METHOD PUBLIC DoPlanning : BOOL
VAR_INPUT
	count : UDINT;
END_VAR
VAR
	i, j  : INT;
END_VAR
IF count = 0 THEN
	isFinished := FALSE;
	Initialize();
END_IF

IF RequireRepeateBlegCenter=TRUE AND BlegCenterFinished=TRUE AND state=BlegCenter THEN
	state:=ready;
    RequireBlegCenter:=TRUE;
	RequireRepeateBlegCenter:=FALSE;
END_IF
IF RequireRepeateStoneRot=TRUE AND StoneRotFinished=TRUE AND state=StoneRot THEN
	state:=MlegRollB;
    MlegRollBFinished:=TRUE;
    RequireStoneRot:=TRUE;
	RequireRepeateStoneRot:=FALSE;
END_IF

IF RequireRepeateBodyPosAdjust=TRUE AND state=BodyPosAdjust AND BodyPosAdjustFinished=TRUE THEN
	state:=ReduceHeight;
    ReduceHeightFinished:=TRUE; 
	RequireBodyPosAdjust:=TRUE;
	RequireRepeateBodyPosAdjust:=FALSE;
END_IF
IF RequireRepeateBLegPosAdjust=TRUE AND state=BLegPosAdjust AND BLegPosAdjustFinished=TRUE THEN
	state:=BodyPosAdjust;
    BodyPosAdjustFinished:=TRUE; 
	RequireBLegPosAdjust:=TRUE;
	RequireRepeateBLegPosAdjust:=FALSE;
END_IF

IF RequireRepeateSearchPedal=TRUE AND state=SearchPedal AND SearchPedalFinished=TRUE THEN
	state:=BLegPosAdjust;
    BLegPosAdjustFinished:=TRUE; 
	RequireSearchPedal:=TRUE;
	RequireRepeateSearchPedal:=FALSE;
END_IF

IF RequireRepeateArmControl=TRUE AND state=ArmControl AND ArmControlFinished=TRUE THEN
	state:=SearchPedal;
    SearchPedalFinished:=TRUE; 
	RequireArmControl:=TRUE;
	RequireRepeateArmControl:=FALSE;
END_IF

IF RequireRepeateOrientAdjust=TRUE AND state=OrientAdjust AND OrientAdjustFinished=TRUE THEN
	state:=ArmControl;
    ArmControlFinished:=TRUE; 
	RequireOrientAdjust:=TRUE;
	RequireRepeateOrientAdjust:=FALSE;
END_IF

StateMachine();
TrjPlanning();

IF quit_flag THEN
	isFinished := TRUE;
	quit_flag := FALSE;
	AC_visual_start:=AC_visual_start;
	
RequireAddHeightFromWalk:=FALSE;
RequireBlegCenter:=FALSE;
RequireMlegRollA:=FALSE;
RequireFlegRotA:=FALSE;
RequireReduceHeight:=FALSE;	
RequireBodyPosAdjust:=FALSE;
RequireBLegPosAdjust:=FALSE;
RequireSearchPedal:=FALSE;
RequireArmControl:=FALSE;
RequireOrientAdjust:=FALSE;
RequireMlegRollB:=FALSE;	
RequireStoneRot:=FALSE;		
RequireLiftMleg:=FALSE;
RequireSpeedUp:=FALSE;
RequireSlide:=FALSE;
RequirePushReleaseBall:=FALSE;
RequireSpeedDown:=FALSE;
RequireBLegRecovery:=FALSE;
RequireMlegRollC:=FALSE;
RequireAddHeight:=FALSE;
RequireFlegRotB:=FALSE;
RequireRecovery:=FALSE;
RequireReduceHeightB:=FALSE;

AddHeightFromWalkFinished:=FALSE;
BlegCenterFinished:=FALSE;
MlegRollAFinished:=FALSE;
FlegRotAFinished:=FALSE;
ReduceHeightFinished:=FALSE;
BodyPosAdjustFinished:=FALSE;
BLegPosAdjustFinished:=FALSE;
SearchPedalFinished:=FALSE;
ArmControlFinished:=FALSE;
OrientAdjustFinished:=FALSE;
MlegRollBFinished:=FALSE;
StoneRotFinished:=FALSE;
LiftMlegFinished:=FALSE;
SpeedUpFinished:=FALSE;
SlideFinished:=FALSE;
PushReleaseBallFinished:=FALSE;
SpeedDownFinished:=FALSE;
BLegRecoveryFinished:=FALSE;
MlegRollCFinished:=FALSE;
AddHeightFinished:=FALSE;
FlegRotBFinished:=FALSE;
CurlingGaitFinished:=FALSE;
RecoveryFinished:=FALSE;
ReduceHeightBFinished:=FALSE;
ReadyFinished:=FALSE;
IsCurlingFinished:=FALSE;
CurlingGaitFinished:=FALSE;
	
	RequireRepeateBlegCenter:=FALSE;
	RequireRepeateBodyPosAdjust:=FALSE;
	RequireRepeateSearchPedal:=FALSE;
	RequireRepeateBLegPosAdjust:=FALSE;
	RequireRepeateOrientAdjust:=FALSE;
	RequireRepeateStoneRot:=FALSE;
END_IF
END_METHOD

METHOD PUBLIC Initialize : BOOL
VAR_INPUT
END_VAR
VAR
	i, j : INT;
	
	leg_pos    : ARRAY[0..2] OF LREAL;
	
	Rb : Mat3;
	hip_pos_j  : Vec3;
	leg_pos_wrt_com : Vec3;
	
END_VAR
Rleg[0]:=SetMat3(1,0,0,0,0,-1,0,1,0);
Rleg[1]:=SetMat3(-1,0,0,0,0,1,0,1,0,);
Rleg[2]:=SetMat3(-1,0,0,0,0,1,0,1,0);
Rleg[3]:=SetMat3(-1,0,0,0,0,1,0,1,0);
Rleg[4]:=SetMat3( -1,0,0,0,0,1,0,1,0);
Rleg[5]:=SetMat3(1,0,0,0,0,-1,0,1,0);

state:=Ready;
ReadyFinished:=true;
quit_flag  := FALSE;
gait_cycle := 0;
AC_visual_start:=FALSE;

IF gvl.taskChooseId=0 THEN //击打
	gvl.target_vel_init:=2;
	gvl.PushVelocityIn_init:=2.3;
	gvl.stone_rot_vel_init:=-60;
	gvl.slideTimeIn_init:=0.3;
	gvl.PushFinishDurationTimeIn_init:=1;
ELSE //进营
	gvl.target_vel_init:=2;
	gvl.PushVelocityIn_init:=1.15;
	gvl.stone_rot_vel_init:=30;	
	gvl.slideTimeIn_init:=0.3;
	gvl.PushFinishDurationTimeIn_init:=1;
END_IF

gvl.adjust_angle_degree:=gvl.adjust_angle_degree_init;
gvl.target_vel:=gvl.target_vel_init;
gvl.stone_rot_vel:=gvl.stone_rot_vel_init;//rpm
gvl.PushVelocityIn:=gvl.PushVelocityIn_init;
gvl.BPA_adjust_angle_degree:=gvl.BPA_adjust_angle_degree_init;//degree
gvl.BPA_adjust_x:=gvl.BPA_adjust_x_init;
gvl.BPA_adjust_y:=gvl.BPA_adjust_y_init;
gvl.BLPA_adjust_distance_desire:=gvl.BLPA_adjust_distance_desire_init;	
gvl.curlingPushModel:=gvl.curlingPushModel_init;	
gvl.PushFinishDurationTimeIn:=gvl.PushFinishDurationTimeIn_init;
gvl.slideTimeIn:=gvl.slideTimeIn_init;
gvl.ArmRetractControl:=gvl.ArmRetractControl_init;
gvl.AC_AngleDegIn:=gvl.AC_AngleDegIn_init;	

// control button for each state, need be commented out at actual environment
RequireAddHeightFromWalk:=FALSE;
RequireBlegCenter:=FALSE;
RequireMlegRollA:=FALSE;
RequireFlegRotA:=FALSE;
RequireReduceHeight:=FALSE;	
RequireBodyPosAdjust:=FALSE;
RequireBLegPosAdjust:=FALSE;
RequireSearchPedal:=FALSE;
RequireArmControl:=FALSE;
RequireOrientAdjust:=FALSE;
RequireMlegRollB:=FALSE;	
RequireStoneRot:=FALSE;		
RequireLiftMleg:=FALSE;
RequireSpeedUp:=FALSE;
RequireSlide:=FALSE;
RequirePushReleaseBall:=FALSE;
RequireSpeedDown:=FALSE;
RequireBLegRecovery:=FALSE;
RequireMlegRollC:=FALSE;
RequireAddHeight:=FALSE;
RequireFlegRotB:=FALSE;
RequireRecovery:=FALSE;
RequireReduceHeightB:=FALSE;

AddHeightFromWalkFinished:=FALSE;
BlegCenterFinished:=FALSE;
MlegRollAFinished:=FALSE;
FlegRotAFinished:=FALSE;
ReduceHeightFinished:=FALSE;
BodyPosAdjustFinished:=FALSE;
BLegPosAdjustFinished:=FALSE;
SearchPedalFinished:=FALSE;
ArmControlFinished:=FALSE;
OrientAdjustFinished:=FALSE;
MlegRollBFinished:=FALSE;
StoneRotFinished:=FALSE;
LiftMlegFinished:=FALSE;
SpeedUpFinished:=FALSE;
SlideFinished:=FALSE;
PushReleaseBallFinished:=FALSE;
SpeedDownFinished:=FALSE;
BLegRecoveryFinished:=FALSE;
MlegRollCFinished:=FALSE;
AddHeightFinished:=FALSE;
FlegRotBFinished:=FALSE;
CurlingGaitFinished:=FALSE;
RecoveryFinished:=FALSE;
ReduceHeightBFinished:=FALSE;

RequireRepeateBlegCenter:=FALSE;
RequireRepeateBodyPosAdjust:=FALSE;
RequireRepeateBLegPosAdjust:=FALSE;
RequireRepeateSearchPedal:=FALSE;
RequireRepeateArmControl:=FALSE;
RequireRepeateOrientAdjust:=FALSE;
RequireRepeateStoneRot:=FALSE;

// bodyRot
delta_t:=1.0/gvl.SampleRate;//sample time
SetTargetValue(GVL.adjust_angle_degree,GVL.target_vel,GVL.stone_rot_vel);
IsReady:=true;

FOR i := 0 TO 5 DO
	FOR j := 0 TO 2 DO
		(*IF ABS(gvl.jntLastRefPos[i, j] - gvl.jntActualPos[i, j]) < gvl.curling_threshold_value THEN
			joint_ref_pos_init[i].data[j] := gvl.jntLastRefPos[i, j];
		ELSE
			joint_ref_pos_init[i].data[j] := gvl.jntActualPos[i, j];
		END_IF*)
		joint_ref_pos_init[i].data[j] := gvl.jntLastRefPos[i, j];
		jointPosLast[i,j]:=joint_ref_pos_init[i].data[j];
	END_FOR
END_FOR

sum_height := 0;
FOR j := 0 TO 5 DO
	// FK
	gvl.legCtrl[j].ForwardKinetics(motorAngles := joint_ref_pos_init[j].data, legIndex:=j, tipPosition => leg_pos);
	leg_ref_pos_init_wrt_hip[j] := SetVec3(leg_pos[0], leg_pos[1], leg_pos[2]);
	sum_height := sum_height - leg_ref_pos_init_wrt_hip[j].data[1];
END_FOR
body_ref_pos_init := SetVec3(0, 0, sum_height/6.0);
body_ref_ang_init := SetVec3(0, 0, 0);                            

FOR j := 0 TO 5 DO
	fbRotMat(yaw := body_ref_ang_init.data[2],
             pitch := body_ref_ang_init.data[1],
             roll := body_ref_ang_init.data[0],
             rm => Rb );
	hip_pos_j := SetVec3(hip_pos[j, 0], hip_pos[j, 1], hip_pos[j, 2]);
	leg_pos_wrt_com := VecAdd(MatMulVec(Rleg[j], leg_ref_pos_init_wrt_hip[j]), hip_pos_j);
    leg_ref_pos_init[j] := VecAdd(body_ref_pos_init, MatMulVec(Rb, leg_pos_wrt_com));
END_FOR

body_ref_pos := body_ref_pos_init;
body_ref_ang := body_ref_ang_init;
leg_ref_pos := leg_ref_pos_init;
leg_ref_pos_wrt_hip := leg_ref_pos_init_wrt_hip;
leg_ref_pos_last:=leg_ref_pos;

FOR i := 0 TO 5 DO
	FOR j := 0 TO 2 DO
		jointPosTarget[i, j] := joint_ref_pos_init[i].data[j];
		jointVelTarget[i, j] := 0;
		jointFceTarget[i, j] := 0;
	END_FOR
END_FOR
END_METHOD

METHOD PUBLIC isPedal : BOOL
VAR_INPUT
		legIndex:INT;
END_VAR
IF ABS(gvl.tipActualFce[legIndex,0])>30 THEN //10 need be calibrated40-->35
	isPedal:=TRUE;
ELSE
	isPedal:=FALSE;
END_IF
END_METHOD

METHOD PUBLIC isStone : BOOL
VAR_INPUT
	legIndex:INT;
END_VAR
IF ABS(gvl.tipActualFce[legIndex,2])>50 THEN //10 need be calibrated
	isStone:=TRUE;
ELSE
	isStone:=FALSE;
END_IF
END_METHOD

METHOD PUBLIC SetTargetValue : BOOL
VAR_INPUT
	in_adjust_angle_degree:LREAL:=0;//unit:degree
	in_target_vel:LREAL:=0;//unit:m/s
	in_stone_rot_vel:LREAL:=0;//unit:rpm
END_VAR
adjust_angle_rad:=in_adjust_angle_degree*pi/180;
target_vel:=in_target_vel;
stone_rot_vel:=in_stone_rot_vel/60*2*pi;
END_METHOD

METHOD PUBLIC StateMachine : BOOL
VAR_INPUT
END_VAR

VAR
	i: INT;
	j: INT;
	RotRadius: LREAL;
END_VAR
IF state=ready AND RequireAddHeightFromWalk=TRUE THEN
	state:=AddHeightFromWalk;
	IsReady:=FALSE;
	IsAddHeightFromWalk:=TRUE;
	RequireAddHeightFromWalk:=FALSE;
	body_ref_pos_enter := body_ref_pos;
	body_ref_ang_enter := body_ref_ang;
	leg_ref_pos_enter := leg_ref_pos;
	EnterAddHeightFromWalkCount:=gait_cycle;
	AddHeightFromWalkFinished:=FALSE;
	AHFW_body_target_pos:=body_ref_pos_enter;
	AHFW_body_target_pos.data[2]:=AHFW_body_target_pos.data[2]+compensateDistance;	

ELSIF state=AddHeightFromWalk AND RequireBlegCenter=TRUE THEN
	state:=BlegCenter;
	IsAddHeightFromWalk:=FALSE;
	IsBlegCenter:=TRUE;
	RequireBlegCenter:=FALSE;
	body_ref_pos_enter := body_ref_pos;
	body_ref_ang_enter := body_ref_ang;
	leg_ref_pos_enter := leg_ref_pos;
	EnterBlegCenterCount:=gait_cycle;
	IsLeg0Move:=TRUE;
	BlegCenterFinished:=FALSE;
	FOR i:=0 TO 1 DO
		FOR j:=0 TO 2 DO
			BlegCenter_BJntStart[i].data[j]:=jointPosLast[Mapping05[i],j];
		END_FOR
	END_FOR
ELSIF state=BlegCenter AND BlegCenterFinished=TRUE AND RequireMlegRollA=TRUE THEN
	state:=MlegRollA;
	IsBlegCenter:=FALSE;
	IsMlegRollA:=TRUE;
	requireMlegRollA:=FALSE;
	body_ref_pos_enter := body_ref_pos;
	body_ref_ang_enter := body_ref_ang;
	leg_ref_pos_enter := leg_ref_pos;
	EnterMlegRollACount:=gait_cycle;
	MlegRollAFinished:=FALSE;
	FOR i:=0 TO 1 DO
		FOR j:=0 TO 2 DO
			MlegRollA_MJntStart[i].data[j]:=jointPosLast[Mapping14[i],j];
		END_FOR
	END_FOR
ELSIF state=MlegRollA AND MlegRollAFinished=TRUE AND RequireFlegRotA=TRUE THEN
	state:=FlegRotA;
	IsMlegRollA:=FALSE;
	IsFlegRotA:=TRUE;
	requireFlegRotA:=FALSE;
	body_ref_pos_enter := body_ref_pos;
	body_ref_ang_enter := body_ref_ang;
	leg_ref_pos_enter := leg_ref_pos;
	EnterFlegRotACount:=gait_cycle;
	FlegRotAFinished:=FALSE;
	FOR i:=0 TO 1 DO
		FOR j:=0 TO 2 DO
			FlegRotA_FJntStart[i].data[j]:=jointPosLast[Mapping23[i],j];
		END_FOR
	END_FOR
ELSIF state=FlegRotA AND FlegRotAFinished=TRUE AND RequireReduceHeight=TRUE THEN
	state:=ReduceHeight;
	IsFlegRotA:=FALSE;
	IsReduceHeight:=TRUE;
	requireReduceHeight:=FALSE;
	body_ref_pos_enter := body_ref_pos;
	body_ref_ang_enter := body_ref_ang;
	leg_ref_pos_enter := leg_ref_pos;
	EnterReduceHeightCount:=gait_cycle;
	body_target_pos:=body_ref_pos_enter;
	body_target_pos.data[2]:=targetHeight;
	ReduceHeightFinished:=FALSE;
	FOR i:=0 TO 1 DO
		FOR j:=0 TO 2 DO
			ReduceHeight_FJntRef[i].data[j]:=jointPosLast[Mapping23[i],j];
		END_FOR
	END_FOR
ELSIF state=ReduceHeight AND ReduceHeightFinished=TRUE AND RequireBodyPosAdjust=TRUE THEN
	state:=BodyPosAdjust;
	IsReduceHeight:=FALSE;
	IsBodyPosAdjust:=TRUE;
	requireBodyPosAdjust:=FALSE;
	body_ref_pos_enter := body_ref_pos;
	body_ref_ang_enter := body_ref_ang;
	leg_ref_pos_enter := leg_ref_pos;
	EnterBodyPosAdjustCount:=gait_cycle;
	BodyPosAdjustFinished:=FALSE;		
	FOR i:=0 TO 1 DO
		FOR j:=0 TO 2 DO
			BPA_FJntRef[i].data[j]:=jointPosLast[Mapping23[i],j];
			BPA_MJntExtend[i,j]:=jointPosLast[Mapping14[i],j];
			BPA_BJntExtend[i,j]:=jointPosLast[Mapping05[i],j];
		END_FOR
		BPA_MJntExtract[i,0]:=BPA_MJntExtend[i,0];
		BPA_MJntExtract[i,1]:=BPA_MJntExtend[i,1]-10*pi/180.0;
		BPA_MJntExtract[i,2]:=BPA_MJntExtend[i,2]+10*pi/180.0;
		BPA_BJntExtract[i,0]:=BPA_BJntExtend[i,0];
		BPA_BJntExtract[i,1]:=BPA_BJntExtend[i,1]-10*pi/180.0;
		BPA_BJntExtract[i,2]:=BPA_BJntExtend[i,2]+10*pi/180.0;
	END_FOR	
	FOR i:=0 TO 2 DO
		BPA_RotCenter1.data[i]:=0.5*(leg_ref_pos_enter[0].data[i]+leg_ref_pos_enter[5].data[i]);
	END_FOR	
	BPA_BodyPosStart:=body_ref_pos_enter;
	BPA_BodyAngStart:=body_ref_ang_enter;	
	RotRadius:=SQRT((BPA_BodyPosStart.data[0]-BPA_RotCenter1.data[0])*(BPA_BodyPosStart.data[0]-BPA_RotCenter1.data[0])+
				(BPA_BodyPosStart.data[1]-BPA_RotCenter1.data[1])*(BPA_BodyPosStart.data[1]-BPA_RotCenter1.data[1]));	
	BPA_AngRad:=GVL.BPA_adjust_angle_degree*pi/180;
	BPA_x:=gvl.BPA_adjust_x;
	BPA_y:=gvl.BPA_adjust_y;
	BPA_BodyPoseEnd.data[0]:=BPA_RotCenter1.data[0]+RotRadius*COS(BPA_AngRad+BPA_BodyAngStart.data[2])+BPA_x;
	BPA_BodyPoseEnd.data[1]:=BPA_RotCenter1.data[1]+RotRadius*SIN(BPA_AngRad+BPA_BodyAngStart.data[2])+BPA_y;
	BPA_BodyPoseEnd.data[2]:=body_ref_pos_enter.data[2];
	BPA_BodyAngEnd:=BPA_BodyAngStart;
	BPA_BodyAngEnd.data[2]:=BPA_BodyAngStart.data[2]+BPA_AngRad;	
ELSIF state=BodyPosAdjust AND BodyPosAdjustFinished=TRUE AND RequireBLegPosAdjust=TRUE THEN
	state:=BLegPosAdjust;
	IsBodyPosAdjust:=FALSE;
	IsBLegPosAdjust:=TRUE;
	requireBLegPosAdjust:=FALSE;
	body_ref_pos_enter := body_ref_pos;
	body_ref_ang_enter := body_ref_ang;
	leg_ref_pos_enter := leg_ref_pos;
	EnterBLegPosAdjustCount:=gait_cycle;
	BLegPosAdjustFinished:=FALSE;	
	
	BLPA_tgtLegPos:=leg_ref_pos_enter;
	BLPA_adjust_distance:=gvl.BLPA_adjust_distance_desire;
	FOR i:=0 TO 1 DO
		FOR j:=0 TO 1 DO
			BLPA_tgtLegPos[Mapping05[i]].data[j]:=leg_ref_pos_enter[Mapping05[i]].data[j]+BLPA_adjust_distance[i,j];
		END_FOR
	END_FOR
	
ELSIF state=BLegPosAdjust AND BLegPosAdjustFinished=TRUE AND RequireSearchPedal=TRUE THEN
	state:=SearchPedal;
	IsBLegPosAdjust:=FALSE;
	IsSearchPedal:=TRUE;
	requireSearchPedal:=FALSE;
	body_ref_pos_enter := body_ref_pos;
	body_ref_ang_enter := body_ref_ang;
	leg_ref_pos_enter := leg_ref_pos;
	EnterSearchPedalCount:=gait_cycle;
	SearchPedalFinished:=FALSE;	
	SP_RBLegSearching:=TRUE;SP_LBLegSearching:=FALSE;
	SP_BLegSearchFinished[0]:=FALSE;SP_BLegSearchFinished[1]:=FALSE;
	SP_PedalSearched[0]:=FALSE;SP_PedalSearched[1]:=FALSE;
	SP_EnterSubSearchCount[0]:=gait_cycle;SP_EnterSubSearchCount[1]:=gait_cycle;
	SP_EnterSubSearchDecreaseCount[0]:=gait_cycle;SP_EnterSubSearchDecreaseCount[1]:=gait_cycle;
	FOR i:=0 TO 1 DO
		FOR j:=0 TO 2 DO
			SP_BJntStart[i].data[j]:=jointPosLast[Mapping05[i],j];
		END_FOR
		gvl.legCtrl[Mapping05[i]].ForwardKinetics(motorAngles:=SP_BJntStart[i].data , legIndex:=Mapping05[i] , tipPosition=>SP_BPosStartWrtHip[i].data );
	END_FOR
ELSIF state=SearchPedal AND SearchPedalFinished=TRUE AND RequireArmControl=TRUE THEN
	state:=ArmControl;
	IsSearchPedal:=FALSE;
	IsArmControl:=TRUE;
	requireArmControl:=FALSE;
	body_ref_pos_enter := body_ref_pos;
	body_ref_ang_enter := body_ref_ang;
	leg_ref_pos_enter := leg_ref_pos;
	EnterArmControlCount:=gait_cycle;
	ArmControlFinished:=FALSE;	
	
	AC_AngleDeg:=gvl.AC_AngleDegIn;
	AC_AngleRad:=AC_AngleDeg*pi/180;
	AC_Velocity:=AC_AngleRad/AC_time;
	AC_extend:=TRUE;
	AC_retract:=FALSE;
	AC_wait:=FALSE;
	AC_EnterExtendCount:=gait_cycle;
	AC_EnterRetractCount:=gait_cycle;
	AC_visual_start:=false;
	

ELSIF state=ArmControl AND ArmControlFinished=TRUE AND RequireOrientAdjust=TRUE THEN
	state:=OrientAdjust;
	IsArmControl:=FALSE;
	IsOrientAdjust:=TRUE;
	requireOrientAdjust:=FALSE;
	body_ref_pos_enter := body_ref_pos;
	body_ref_ang_enter := body_ref_ang;
	leg_ref_pos_enter := leg_ref_pos;
	EnterOrientAdjustCount:=gait_cycle;
	OrientAdjustFinished:=FALSE;	
	FOR i:=0 TO 1 DO
		FOR j:=0 TO 2 DO
			OA_FJntRef[i].data[j]:=jointPosLast[Mapping23[i],j];
			OA_MJntExtend[i,j]:=jointPosLast[Mapping14[i],j];
		END_FOR
		OA_MJntExtract[i,0]:=OA_MJntExtend[i,0];
		OA_MJntExtract[i,1]:=OA_MJntExtend[i,1]-10*pi/180.0;
		OA_MJntExtract[i,2]:=OA_MJntExtend[i,2]+10*pi/180.0;
	END_FOR
	FOR i:=0 TO 2 DO
		OA_RotCenter1.data[i]:=0.5*(leg_ref_pos_enter[0].data[i]+leg_ref_pos_enter[5].data[i]);
	END_FOR
	OA_BodyPosStart:=body_ref_pos_enter;
	OA_BodyAngStart:=body_ref_ang_enter;
	RotRadius:=SQRT((OA_BodyPosStart.data[0]-OA_RotCenter1.data[0])*(OA_BodyPosStart.data[0]-OA_RotCenter1.data[0])+
               (OA_BodyPosStart.data[1]-OA_RotCenter1.data[1])*(OA_BodyPosStart.data[1]-OA_RotCenter1.data[1]));
	adjust_angle_rad:=GVL.adjust_angle_degree*pi/180;
	OA_BodyPoseEnd.data[0]:=OA_RotCenter1.data[0]+RotRadius*COS(adjust_angle_rad+OA_BodyAngStart.data[2]);
	OA_BodyPoseEnd.data[1]:=OA_RotCenter1.data[1]+RotRadius*SIN(adjust_angle_rad+OA_BodyAngStart.data[2]);
	OA_BodyPoseEnd.data[2]:=body_ref_pos_enter.data[2];
	OA_BodyAngEnd:=OA_BodyAngStart;
	OA_BodyAngEnd.data[2]:=OA_BodyAngStart.data[2]+adjust_angle_rad;
ELSIF state=OrientAdjust AND OrientAdjustFinished=TRUE AND RequireMlegRollB=TRUE THEN
	state:=MlegRollB;
	IsOrientAdjust:=FALSE;
	IsMlegRollB:=TRUE;
	requireMlegRollB:=FALSE;
	body_ref_pos_enter := body_ref_pos;
	body_ref_ang_enter := body_ref_ang;
	leg_ref_pos_enter := leg_ref_pos;
	EnterMlegRollBCount:=gait_cycle;
	FOR i:=0 TO 1 DO
		FOR j:=0 TO 2 DO
			MlegRollB_MJntStart[i].data[j]:=jointPosLast[Mapping14[i],j];
		END_FOR
	END_FOR	
ELSIF state=MlegRollB AND MlegRollBFinished=TRUE AND RequireStoneRot=TRUE THEN
	state:=StoneRot;
	stone_rot_vel:=GVL.stone_rot_vel/60*2*pi;
	IsMlegRollB:=FALSE;
	IsStoneRot:=TRUE;
	requireStoneRot:=FALSE;
	body_ref_pos_enter := body_ref_pos;
	body_ref_ang_enter := body_ref_ang;
	leg_ref_pos_enter := leg_ref_pos;
	EnterStoneRotCount:=gait_cycle;
	StoneRotFinished:=FALSE;
	SetColide:=FALSE;
	StoneRotSubState[0]:=FALSE;
	StoneRotSubState[1]:=FALSE;
	FOR i:=0 TO 1 DO
		FOR j:=0 TO 2 DO
			StoneRot_FJntStart[i].data[j]:=jointPosLast[Mapping23[i],j];
		END_FOR
	END_FOR
ELSIF state=StoneRot AND StoneRotFinished=TRUE AND  RequireLiftMleg=TRUE THEN
	state:=LiftMleg;
	IsStoneRot:=FALSE;
	IsLiftMleg:=TRUE;
	requireLiftMleg:=FALSE;	
	body_ref_pos_enter := body_ref_pos;
	body_ref_ang_enter := body_ref_ang;
	leg_ref_pos_enter := leg_ref_pos;
	EnterLiftMlegCount:=gait_cycle;
	LiftMlegFinished:=FALSE;
	FOR i:=0 TO 1 DO
		FOR j:=0 TO 2 DO
			LiftMleg_MJntStart[i].data[j]:=jointPosLast[Mapping14[i],j];
		END_FOR
	END_FOR	
ELSIF state=LiftMleg AND LiftMlegFinished=TRUE AND RequireSpeedUp=TRUE THEN
	state:=SpeedUp;
	IsLiftMleg:=FALSE;
	IsSpeedUp:=TRUE;
	requireSpeedUp:=FALSE;	
	IF ABS(GVL.target_vel)<=0.5 THEN
		GVL.target_vel:=0.5;
	END_IF
	target_vel:=GVL.target_vel;
	body_ref_pos_enter := body_ref_pos;
	body_ref_ang_enter := body_ref_ang;
	leg_ref_pos_enter := leg_ref_pos;
	EnterSpeedUpCount:=gait_cycle;
	SpeedUpFinished:=FALSE;
	FOR i:=0 TO 1 DO
		FOR j:=0 TO 2 DO
			SpeedUp_MJntRef[i].data[j]:=jointPosLast[Mapping14[i],j];
			SpeedUp_FJntRef[i].data[j]:=jointPosLast[Mapping23[i],j];
			SpeedUp_BJntStart[i].data[j]:=jointPosLast[Mapping05[i],j];
		END_FOR
		gvl.legCtrl[Mapping05[i]].ForwardKinetics(motorAngles:=SpeedUp_BJntStart[i].data , legIndex:=Mapping05[i] , tipPosition=>SpeedUp_BPosWrtHipStart[i].data );
	END_FOR	
	CurrentBLegMaxDistance:=MAX(ABS(SpeedUp_BPosWrtHipStart[0].data[0]),ABS(SpeedUp_BPosWrtHipStart[1].data[0]));
	Distance_x_total:=0.85-CurrentBLegMaxDistance;
	IF Distance_x_total<0 THEN
		quit_flag:=TRUE;
		SpeedUpFinished:=true;
	END_IF
	
	SpeedUpSubState:=SpeedUpAS;
	EnterSpeedUpASCount:=gait_cycle;

	Distance_x_AS:=Distance_x_total-Distance_x_DS-target_vel*Time_CS;
	Time_AS:=2.0*Distance_x_AS/target_vel;
ELSIF state=SpeedUp AND SpeedUpFinished=TRUE AND RequireSlide=TRUE THEN
	state:=Slide;
	IsSpeedUp:=FALSE;
	IsSlide:=TRUE;
	requireSlide:=FALSE;	
	body_ref_pos_enter := body_ref_pos;
	body_ref_ang_enter := body_ref_ang;
	leg_ref_pos_enter := leg_ref_pos;
	EnterSlideCount:=gait_cycle;
	SlideFinished:=FALSE;
	slideTime:=gvl.slideTimeIn;
ELSIF state=Slide AND SlideFinished=TRUE AND RequirePushReleaseBall=TRUE THEN
	state:=PushReleaseBall;
	IsSlide:=FALSE;
	IsPushReleaseBall:=TRUE;
	RequirePushReleaseBall:=FALSE;
	body_ref_pos_enter := body_ref_pos;
	body_ref_ang_enter := body_ref_ang;
	leg_ref_pos_enter := leg_ref_pos;
	EnterPushReleaseBallCount:=gait_cycle;
	PushReleaseBallFinished:=FALSE;
	PushFinishDurationTime:=gvl.PushFinishDurationTimeIn;
	FOR i:=0 TO 1 DO
		FOR j:=0 TO 2 DO
			PushReleaseBall_FJntStart[i].data[j]:=jointPosLast[Mapping23[i],j];
		END_FOR
		gvl.legCtrl[Mapping23[i]].ForwardKinetics(motorAngles:=PushReleaseBall_FJntStart[i].data , legIndex:=Mapping23[i] , tipPosition=>PushReleaseBall_FPosStartWrtHip[i].data );
	END_FOR
	IF ABS(gvl.PushVelocityIn)<=0.1 THEN
		gvl.PushVelocityIn:=0;
	END_IF
	PushVelocity:=gvl.PushVelocityIn;
	PushDistance:=PRDistance_x_total-DecVelDistance-PRConstVelTime*PushVelocity;
	PRConstVelDistance:=PRConstVelTime*PushVelocity;
	PushTime:=PushDistance*2/PushVelocity;
	
ELSIF state=PushReleaseBall AND PushReleaseBallFinished=TRUE AND RequireSpeedDown=TRUE THEN
	state:=SpeedDown;
	IsPushReleaseBall:=FALSE;
	IsSpeedDown:=TRUE;
	RequireSpeedDown:=FALSE;
	body_ref_pos_enter := body_ref_pos;
	body_ref_ang_enter := body_ref_ang;
	leg_ref_pos_enter := leg_ref_pos;
	EnterSpeedDownCount:=gait_cycle;
	SpeedDownFinished:=FALSE;
	FOR i:=0 TO 1 DO
		FOR j:=0 TO 2 DO
			SpeedDown_MJntStart[i].data[j]:=jointPosLast[Mapping14[i],j];
		END_FOR
	END_FOR
ELSIF state=SpeedDown AND SpeedDownFinished=TRUE AND RequireBLegRecovery=TRUE THEN	
	state:=BLegRecovery;
	IsSpeedDown:=FALSE;
	IsBLegRecovery:=TRUE;
	RequireBLegRecovery:=FALSE;
	body_ref_pos_enter := body_ref_pos;
	body_ref_ang_enter := body_ref_ang;
	leg_ref_pos_enter := leg_ref_pos;
	EnterBLegRecoveryCount:=gait_cycle;
	BLegRecoveryFinished:=FALSE;	
	FOR i:=0 TO 1 DO
		FOR j:=0 TO 2 DO
			BLR_FJntStart[i].data[j]:=jointPosLast[Mapping05[i],j];
		END_FOR
	END_FOR
	
ELSIF state=BLegRecovery AND BLegRecoveryFinished=TRUE AND RequireMlegRollC=TRUE THEN
	state:=MlegRollC;
	IsBLegRecovery:=FALSE;
	IsMlegRollC:=TRUE;
	RequireMlegRollC:=FALSE;
	body_ref_pos_enter := body_ref_pos;
	body_ref_ang_enter := body_ref_ang;
	leg_ref_pos_enter := leg_ref_pos;
	EnterMlegRollCCount:=gait_cycle;
	MlegRollCFinished:=FALSE;	
	FOR i:=0 TO 1 DO
		FOR j:=0 TO 2 DO
			MlegRollC_MJntStart[i].data[j]:=jointPosLast[Mapping14[i],j];
		END_FOR
	END_FOR
ELSIF state=MlegRollC AND MlegRollCFinished=TRUE AND RequireAddHeight=TRUE THEN	
	state:=AddHeight;
	RequireAddHeight:=FALSE;
	IsMlegRollC:=FALSE;
	IsAddHeight:=TRUE;
	body_ref_pos_enter := body_ref_pos;
	body_ref_ang_enter := body_ref_ang;
	leg_ref_pos_enter := leg_ref_pos;
	EnterAddHeightCount:=gait_cycle;
	AddHeightFinished:=FALSE;
	FOR i:=0 TO 1 DO
		FOR j:=0 TO 2 DO
			AddHeight_FJntStart[i].data[j]:=jointPosLast[Mapping23[i],j];
		END_FOR
	END_FOR
	body_target_pos:=body_ref_pos_enter;
	body_target_pos.data[2]:=sum_height/6.0+compensateDistance;
ELSIF state=AddHeight AND AddHeightFinished=TRUE AND RequireFlegRotB=TRUE THEN	
	state:=FlegRotB;
	IsAddHeight:=FALSE;
	IsFlegRotB:=TRUE;
	RequireFlegRotB:=FALSE;
	body_ref_pos_enter := body_ref_pos;
	body_ref_ang_enter := body_ref_ang;
	leg_ref_pos_enter := leg_ref_pos;
	EnterFlegRotBCount:=gait_cycle;
	FlegRotBFinished:=FALSE;
	FOR i:=0 TO 1 DO
		FOR j:=0 TO 2 DO
			FlegRotB_FJntStart[i].data[j]:=jointPosLast[Mapping23[i],j];
		END_FOR
	END_FOR
ELSIF state=FlegRotB AND FlegRotBFinished=TRUE AND RequireRecovery=TRUE THEN	
	state:=Recovery;
	IsFlegRotB:=FALSE;
	IsRecovery:=TRUE;
	RequireRecovery:=FALSE;	
	body_ref_pos_enter := body_ref_pos;
	body_ref_ang_enter := body_ref_ang;
	leg_ref_pos_enter := leg_ref_pos;
	EnterRecoveryCount:=gait_cycle;
	RecoveryFinished:=FALSE;	
	RcJointPosStart:=jointPosLast;
	
ELSIF state=Recovery AND RecoveryFinished=TRUE AND RequireReduceHeightB=TRUE THEN	
	state:=ReduceHeightB;
	IsRecovery:=FALSE;
	IsReduceHeightB:=TRUE;
	RequireReduceHeightB:=FALSE;	
	body_ref_pos_enter := body_ref_pos;
	body_ref_ang_enter := body_ref_ang;
	leg_ref_pos_enter := leg_ref_pos;
	EnterReduceHeightBCount:=gait_cycle;
	ReduceHeightBFinished:=FALSE;	
	RHB_body_target_pos:=body_ref_pos_enter;
	RHB_body_target_pos.data[2]:=RHB_body_target_pos.data[2]-compensateDistance;

ELSIF state=ReduceHeightB AND ReduceHeightBFinished=TRUE THEN	
	IsReduceHeightB:=FALSE;
	IsCurlingFinished:=TRUE;
	state:=CurlingFinished;
	CurlingGaitFinished:=TRUE;
	quit_flag:=TRUE;
END_IF
END_METHOD

METHOD PUBLIC TrjPlanning : BOOL
VAR_INPUT
END_VAR
VAR
	tr : LREAL;
	i, j : INT;
	Rb : Mat3;
	hip_pos_j : Vec3;
	leg_ref_pos_wrt_com_j : Vec3;
	tmp : Vec3;
	tip_pos, tip_vel : Vec3;
	
	body_ref_pos_start : Vec3;
	body_ref_pos_end : Vec3;
	jointTmpPosLast: ARRAY[0..2] OF LREAL;
	body_ref_ang_start: Vec3;
	leg_ref_pos_start: ARRAY [0..5] OF Vec3;
	leg_ref_pos_target: ARRAY [0..5] OF Vec3;
	body_ref_ang_end: Vec3;
	Rb_target2: Mat3;
	Rb_target1: Mat3;
	leg_ref_pos_end: ARRAY [0..5] OF Vec3;
	fbElipseInterpolation:ElipseInterpolation;
	fbHermitInterpolation:HermitInterpolation;
	
	tempTipForce:ARRAY [0..2] OF LREAL;
	temJntActPos:ARRAY [0..2] OF LREAL;
	tempDesJntTrq:ARRAY [0..2] OF LREAL;
END_VAR
gait_cycle := gait_cycle + 1;

IF state=Ready THEN
	body_ref_pos := body_ref_pos_init;
	body_ref_ang := body_ref_ang_init;
	leg_ref_pos := leg_ref_pos_init;
	leg_ref_pos_wrt_hip := leg_ref_pos_init_wrt_hip;
ELSIF state=AddHeightFromWalk THEN
	TrjPlanning_AddHeightFromWalk();
ELSIF state=BlegCenter THEN
	TrjPlanning_BlegCenter();
ELSIF state=MlegRollA THEN
	TrjPlanning_MlegRollA();
ELSIF state=FlegRotA THEN
	TrjPlanning_FlegRotA();
ELSIF state=ReduceHeight THEN
	TrjPlanning_ReduceHeight();
ELSIF state=BodyPosAdjust THEN
	TrjPlanning_BodyPosAdjust();
ELSIF state=BLegPosAdjust THEN
	TrjPlanning_BLegPosAdjust();	
ELSIF state=SearchPedal THEN
	TrjPlanning_SearchPedal();
ELSIF state=ArmControl THEN
	TrjPlanning_ArmControl();
ELSIF state=OrientAdjust THEN	
	TrjPlanning_OrientAdjust();
ELSIF state=MlegRollB THEN
	TrjPlanning_MlegRollB();
ELSIF state=StoneRot THEN
	TrjPlanning_StoneRot();
ELSIF state=LiftMleg THEN
	TrjPlanning_LiftMleg();
ELSIF state=SpeedUp THEN
	TrjPlanning_SpeedUp();
ELSIF state=Slide THEN	
	TrjPlanning_Slide();
ELSIF state=PushReleaseBall THEN
	TrjPlanning_PushReleaseBall();
ELSIF state=SpeedDown THEN	
	TrjPlanning_SpeedDown();
ELSIF state=BLegRecovery THEN	
	TrjPlanning_BLegRecovery();
ELSIF state=MlegRollC THEN	
	TrjPlanning_MlegRollC();
ELSIF state=AddHeight THEN	
	TrjPlanning_AddHeight();
ELSIF state=FlegRotB THEN	
	TrjPlanning_FlegRotB();
ELSIF state=Recovery THEN	
	TrjPlanning_Recovery();	
ELSIF state=ReduceHeightB THEN	
	TrjPlanning_ReduceHeightB();	
END_IF

// transform TO leg local frame AND DO inverse kinematics

FOR j := 0 TO 5 DO
	fbRotMat(
    	yaw := body_ref_ang.data[2], 
		pitch := body_ref_ang.data[1], 
		roll := body_ref_ang.data[0], 
		rm => Rb);
	hip_pos_j := SetVec3(hip_pos[j, 0], hip_pos[j, 1], hip_pos[j, 2]);

	//leg_ref_pos_wrt_com = Rb' * (leg_ref_pos - body_ref_pos)
	leg_ref_pos_wrt_com_j := MatMulVec(
		                         MatTranspose(Rb),
								 VecAdd(
									 leg_ref_pos[j],
									 VecNeg(body_ref_pos)
                                 )
                             );
	// leg_ref_pos_wrt_hip = Rleg' * (leg_ref_pos_wrt_com_j - hip_pos)
	leg_ref_pos_next_wrt_hip[j] := MatMulVec(
		                               MatTranspose(Rleg[j]),
									   VecAdd(
										   leg_ref_pos_wrt_com_j,
										   VecNeg(hip_pos_j)
									   )
								   );
								   
	leg_ref_vel_next_wrt_hip[j] := VecMulNum(VecAdd(leg_ref_pos_next_wrt_hip[j], VecNeg(leg_ref_pos_wrt_hip[j])), DINT_TO_LREAL(gvl.sampleRate));
END_FOR


// mapping to actual joints
FOR j := 0 TO 5 DO
	tmp := leg_ref_pos_next_wrt_hip[leg_index_mapping[j]-1];
	tip_pos := SetVec3(tmp.data[0], tmp.data[1], tmp.data[2]);
	tmp := leg_ref_vel_next_wrt_hip[leg_index_mapping[j]-1];
	tip_vel := SetVec3(tmp.data[0], tmp.data[1], tmp.data[2]);
	FOR i:= 0 TO 2 DO
		jointTmpPosLast[i]:=jointPosLast[j,i];
	END_FOR		
	gvl.legCtrl[j].InversePosAndVel(
		tipPos := tip_pos.data, 
		tipVel := tip_vel.data, 
		refPosLast:=jointTmpPosLast,
		legIndex:=j,
		jntPos => joint_ref_pos[j].data, 
		jntVel => joint_ref_vel[j].data);
	
END_FOR

//generate joint reference torque
FOR i:=0 TO 5 DO
	tempTipForce[0]:=tipForceDesire[i,0];tempTipForce[1]:=tipForceDesire[i,1];tempTipForce[2]:=tipForceDesire[i,2];
	temJntActPos[0]:=gvl.jntActualPos[i,0];temJntActPos[1]:=gvl.jntActualPos[i,1];temJntActPos[2]:=gvl.jntActualPos[i,2];
	gvl.legCtrl[i].DesireDriveForce(fTipDes:=tempTipForce , motorAng:=temJntActPos , legIndex:=i , fDrvDes=>tempDesJntTrq );
	jntTrqDesire[i,0]:=tempDesJntTrq[0];jntTrqDesire[i,1]:=tempDesJntTrq[1];jntTrqDesire[i,2]:=tempDesJntTrq[2];
END_FOR


// link to physical outputs
FOR i := 0 TO 5 DO
	FOR j := 0 TO 2 DO
		jointPosTarget[i, j] := joint_ref_pos[i].data[j];
		jointPosLast[i,j]:=jointPosTarget[i, j] ;
		gvl.jntRefPosLastPlanning[i,j]:=jointPosTarget[i, j] ;
		jointVelTarget[i, j] := joint_ref_vel[i].data[j];
		jointFceTarget[i, j] :=jntTrqDesire[i,j];
	END_FOR
END_FOR

// store refs for next loop
leg_ref_pos_wrt_hip := leg_ref_pos_next_wrt_hip;
leg_ref_pos_last:=leg_ref_pos;

IF gait_cycle > tTotalAll * gvl.sampleRate THEN
	quit_flag := TRUE;
END_IF
END_METHOD

METHOD PUBLIC TrjPlanning_AddHeight : BOOL
VAR_INPUT
END_VAR
VAR
	tr: LREAL;
	i: INT;
	Rb_target1: Mat3;
	temp:vec3;
END_VAR
IF  AddHeightFinished=FALSE AND (gait_cycle-EnterAddHeightCount)<=AddHeightTime*gvl.sampleRate THEN
	body_ref_ang:=body_ref_ang_enter;
	leg_ref_pos:=leg_ref_pos_enter;
	tr  := UDINT_TO_LREAL(gait_cycle - EnterAddHeightCount) / gvl.sampleRate / AddHeightTime;
	fbGetPivot(tNow := tr, tTotal := 1.0, pivot => pvt);
	FOR i:=0 TO 2 DO
		body_ref_pos.data[i]:=(1-pvt)*body_ref_pos_enter.data[i]+pvt*body_target_pos.data[i];
	END_FOR
	
	FOR i:=0 TO 1 DO
		gvl.legCtrl[Mapping23[i]].ForwardKinetics(motorAngles:=AddHeight_FJntStart[i].data , legIndex:=Mapping23[i] , tipPosition=>AddHeight_FPosWrtHip[i].data );
		fbRotMat(yaw := body_ref_ang_enter.data[2], pitch := body_ref_ang_enter.data[1],roll := body_ref_ang_enter.data[0], rm => Rb_target1 );
		temp.data[0]:=hip_pos[Mapping23[i],0];temp.data[1]:=hip_pos[Mapping23[i],1];temp.data[2]:=hip_pos[Mapping23[i],2];
		leg_ref_pos[Mapping23[i]]:= VecAdd( MatMulVec(Rb_target1, VecAdd(temp,MatMulVec(Rleg[Mapping23[i]],AddHeight_FPosWrtHip[i]))),body_ref_pos);
	END_FOR
ELSE
	AddHeightFinished:=TRUE;	
	RequireFlegRotB:=TRUE;//********************************************************************************************************
END_IF
END_METHOD

METHOD PUBLIC TrjPlanning_AddHeightFromWalk : BOOL
VAR_INPUT
END_VAR
VAR
	tr: LREAL;
	i: INT;
	Rb_target1: Mat3;
	temp: vec3;
END_VAR
IF AddHeightFromWalkFinished=FALSE AND (gait_cycle-EnterAddHeightFromWalkCount)<=AHFW_time*gvl.sampleRate THEN
	body_ref_ang:=body_ref_ang_enter;
	leg_ref_pos:=leg_ref_pos_enter;
	tr  := UDINT_TO_LREAL(gait_cycle - EnterAddHeightFromWalkCount) / gvl.sampleRate / AHFW_time;
	fbGetPivot(tNow := tr, tTotal := 1.0, pivot => pvt);
	FOR i:=0 TO 2 DO
		body_ref_pos.data[i]:=(1-pvt)*body_ref_pos_enter.data[i]+pvt*AHFW_body_target_pos.data[i];
	END_FOR
ELSE
	AddHeightFromWalkFinished:=TRUE;
	RequireBlegCenter:=true;
END_IF
END_METHOD

METHOD PUBLIC TrjPlanning_ArmControl : BOOL
VAR_INPUT
END_VAR
IF ArmControlFinished=FALSE THEN
	body_ref_pos:=body_ref_pos_enter;
	body_ref_ang:=body_ref_ang_enter;
	leg_ref_pos:=leg_ref_pos_enter;	
	
	IF AC_extend=TRUE THEN
		AC_wait:=FALSE;
		AC_retract:=FALSE;
		IF (gait_cycle-AC_EnterExtendCount)=1 THEN
			GVL.jogVelocity[20]:=AC_Velocity;
			GVL.jogButton[20]:=TRUE;
		END_IF
		IF (gait_cycle-AC_EnterExtendCount)=LREAL_TO_UDINT(AC_time*gvl.sampleRate) THEN
			GVL.jogVelocity[20]:=0;
			GVL.jogButton[20]:=FALSE;
			GVL.jogStopButton[20]:=TRUE;
		END_IF
		IF (gait_cycle-AC_EnterExtendCount)=LREAL_TO_UDINT((AC_time+0.5)*gvl.sampleRate) THEN
			AC_visual_start:=TRUE;
		END_IF
		IF (gait_cycle-AC_EnterExtendCount)=LREAL_TO_UDINT((AC_time+0.5+2)*gvl.sampleRate) THEN
			AC_visual_start:=FALSE;
			gvl.ArmRetractControl:=TRUE;
		END_IF		
		
	END_IF
	
	IF AC_retract=FALSE AND gvl.ArmRetractControl=TRUE AND (gait_cycle-AC_EnterExtendCount)>=LREAL_TO_UDINT(AC_time*gvl.sampleRate) THEN
		AC_retract:=TRUE;
		AC_visual_start:=FALSE;
		gvl.ArmRetractControl:=FALSE;
		AC_EnterRetractCount:=gait_cycle;
	END_IF
	
	IF AC_retract=TRUE THEN
		AC_extend:=FALSE;
		AC_wait:=FALSE;
		IF (gait_cycle-AC_EnterRetractCount)=1 THEN
			GVL.jogVelocity[20]:=-AC_Velocity;
			GVL.jogButton[20]:=TRUE;
		END_IF	
		IF (gait_cycle-AC_EnterRetractCount)=LREAL_TO_UDINT(AC_time*gvl.sampleRate) THEN
			GVL.jogVelocity[20]:=0;
			GVL.jogButton[20]:=FALSE;
			GVL.jogStopButton[20]:=TRUE;
			ArmControlFinished:=TRUE;
		END_IF
	END_IF
END_IF
END_METHOD

METHOD PUBLIC TrjPlanning_BlegCenter : BOOL
VAR_INPUT
END_VAR
VAR

											 
	(*BC_BPosExtendRefDouble:ARRAY[0..1,0..2] OF LREAL:=[-0.15,-0.3805-0.07-0.01,0,
												       -0.15,-0.3805-0.07-0.01,0];
	BC_BPosExtendRefSingle:ARRAY[0..1,0..2] OF LREAL:=[-0.15,-0.3805-0.07-0.01,-0.05,
												       -0.15,-0.3805-0.07-0.01,0.05];											
	BC_BPosRetractRef:ARRAY[0..1,0..2]      OF LREAL:=[-0.15,-0.3805,0,
												       -0.15,-0.3805,0];*)
													   											 
	BC_BPosExtendRefDouble:ARRAY[0..1,0..2] OF LREAL:=[-0.15,-0.4-0.07-0.01,0.02*1.125,
												       -0.15,-0.4-0.07-0.01,-0.02*1.125];
	BC_BPosExtendRefSingle:ARRAY[0..1,0..2] OF LREAL:=[-0.15,-0.4-0.07-0.01,-0.05,
												       -0.15,-0.4-0.07-0.01,0.05];											
	BC_BPosRetractRef:ARRAY[0..1,0..2]      OF LREAL:=[-0.15,-0.4,0,
												       -0.15,-0.4,0];
												 
	BC_BJntRetractRef:ARRAY[0..1,0..2]      OF LREAL:=[0,180*pi/180,330*pi/180,
                                                       0,180*pi/180,330*pi/180];	
	BC_BJntTargetRef:ARRAY[0..1,0..2]       OF LREAL:=[0*pi/180,190.9254*pi/180, 312.9903*pi/180,
                                                       0*pi/180,190.9254*pi/180, 312.9903*pi/180];//double pedal,[-0.15, -0.3805-0.07-0.01,0]														 
		
	tTotal:lreal;										 
	tNow: LREAL;
	i: INT;
	j: INT;
	tr: LREAL;
	Rb_target1: Mat3;
	temp: vec3;
	tempLeg:ARRAY [0..2] OF LREAL;
	tempJnt:ARRAY [0..2] OF LREAL;
	tempRef:ARRAY [0..2] OF LREAL;
	
	tipForceDesireLegA:	 ARRAY[0..5,0..2] OF LREAL:=[0,-100,0,
													 0,0,0,
													 0,0,0,
													 0,0,0,
													 0,0,0,
													 0,0,0];
	tipForceDesireLegF:	 ARRAY[0..5,0..2] OF LREAL:=[0,0,0,
													 0,0,0,
													 0,0,0,
													 0,0,0,
													 0,0,0,
													 0,-120,0];													 
END_VAR
IF (gait_cycle-EnterBlegCenterCount)=1 THEN
	IF BlegCenterType=0 THEN
		FOR i:=0 TO 1 DO
			tempLeg[0]:=BC_BPosExtendRefDouble[i,0];tempLeg[1]:=BC_BPosExtendRefDouble[i,1];tempLeg[2]:=BC_BPosExtendRefDouble[i,2];
			tempRef[0]:=BC_BJntTargetRef[i,0];tempRef[1]:=BC_BJntTargetRef[i,1];tempRef[2]:=BC_BJntTargetRef[i,2];
			GVL.legCtrl[Mapping05[i]].InverseKinetics(tipPosition:=tempLeg , refPosLast:=tempRef , legIndex:=Mapping05[i] , motorAngles=>tempJnt , isSingular=> );
			BC_BJntTarget[i,0]:=tempJnt[0];BC_BJntTarget[i,1]:=tempJnt[1];BC_BJntTarget[i,2]:=tempJnt[2];
		END_FOR
	ELSE
		FOR i:=0 TO 1 DO
			tempLeg[0]:=BC_BPosExtendRefSingle[i,0];tempLeg[1]:=BC_BPosExtendRefSingle[i,1];tempLeg[2]:=BC_BPosExtendRefSingle[i,2];
			tempRef[0]:=BC_BJntTargetRef[i,0];tempRef[1]:=BC_BJntTargetRef[i,1];tempRef[2]:=BC_BJntTargetRef[i,2];
			GVL.legCtrl[Mapping05[i]].InverseKinetics(tipPosition:=tempLeg , refPosLast:=tempRef , legIndex:=Mapping05[i] , motorAngles=>tempJnt , isSingular=> );
			BC_BJntTarget[i,0]:=tempJnt[0];BC_BJntTarget[i,1]:=tempJnt[1];BC_BJntTarget[i,2]:=tempJnt[2];
		END_FOR
	END_IF
	FOR i:=0 TO 1 DO
		tempLeg[0]:=BC_BPosRetractRef[i,0];tempLeg[1]:=BC_BPosRetractRef[i,1];tempLeg[2]:=BC_BPosRetractRef[i,2];
		tempRef[0]:=BC_BJntRetractRef[i,0];tempRef[1]:=BC_BJntRetractRef[i,1];tempRef[2]:=BC_BJntRetractRef[i,2];
		GVL.legCtrl[Mapping05[i]].InverseKinetics(tipPosition:=tempLeg , refPosLast:=tempRef , legIndex:=Mapping05[i] , motorAngles=>tempJnt , isSingular=> );
		BC_BJntRetract[i,0]:=tempJnt[0];BC_BJntRetract[i,1]:=tempJnt[1];BC_BJntRetract[i,2]:=tempJnt[2];
	END_FOR	
END_IF

IF (gait_cycle-EnterBlegCenterCount)=(BlegCenterRetractTime+BlegCenterExtendTime)*gvl.sampleRate THEN
	leg_ref_pos_enter:=leg_ref_pos_last;
END_IF
IF IsLeg0Move=FALSE AND (gait_cycle-EnterLeg5MoveCount)=(BlegCenterRetractTime+BlegCenterExtendTime)*gvl.sampleRate THEN
	leg_ref_pos_enter:=leg_ref_pos_last;
END_IF


body_ref_pos:=body_ref_pos_enter;
body_ref_ang:=body_ref_ang_enter;
leg_ref_pos:=leg_ref_pos_enter;
IF BlegCenterFinished=FALSE THEN
	IF IsLeg0Move=TRUE THEN
		IF (gait_cycle-EnterBlegCenterCount)<=BlegCenterRetractTime*gvl.sampleRate THEN
			tr  := UDINT_TO_LREAL(gait_cycle-EnterBlegCenterCount) / gvl.sampleRate / BlegCenterRetractTime;
			fbGetPivot(tNow := tr, tTotal := 1.0, pivot => pvt);
			FOR j:=0 TO 2 DO
				BlegCenter_BJntRef[0].data[j]:=(1-pvt)*BlegCenter_BJntStart[0].data[j]+pvt*(BC_BJntRetract[0,j]);
			END_FOR		
			gvl.legCtrl[Mapping05[0]].ForwardKinetics(motorAngles:=BlegCenter_BJntRef[0].data , legIndex:=Mapping05[0] , tipPosition=>BlegCenter_BPosWrtHip[0].data );
			fbRotMat(yaw := body_ref_ang_enter.data[2], pitch := body_ref_ang_enter.data[1],roll := body_ref_ang_enter.data[0], rm =>  Rb_target1 );
			temp.data[0]:=hip_pos[Mapping05[0],0];temp.data[1]:=hip_pos[Mapping05[0],1];temp.data[2]:=hip_pos[Mapping05[0],2];
			leg_ref_pos[Mapping05[0]]:= VecAdd( MatMulVec(Rb_target1, VecAdd(temp,MatMulVec(Rleg[Mapping05[0]],BlegCenter_BPosWrtHip[0]))),body_ref_pos);
		ELSIF (gait_cycle-EnterBlegCenterCount)<=(BlegCenterRetractTime+BlegCenterExtendTime)*gvl.sampleRate THEN
			tr  := (UDINT_TO_LREAL(gait_cycle-EnterBlegCenterCount) / gvl.sampleRate -BlegCenterRetractTime)/ BlegCenterExtendTime;
			fbGetPivot(tNow := tr, tTotal := 1.0, pivot => pvt);
			FOR j:=0 TO 2 DO
				BlegCenter_BJntRef[0].data[j]:=(1-pvt)*BC_BJntRetract[0,j]+pvt*(BC_BJntTarget[0,j]);
			END_FOR
			gvl.legCtrl[Mapping05[0]].ForwardKinetics(motorAngles:=BlegCenter_BJntRef[0].data , legIndex:=Mapping05[0] , tipPosition=>BlegCenter_BPosWrtHip[0].data );
			fbRotMat(yaw := body_ref_ang_enter.data[2], pitch := body_ref_ang_enter.data[1],roll := body_ref_ang_enter.data[0], rm =>  Rb_target1 );
			temp.data[0]:=hip_pos[Mapping05[0],0];temp.data[1]:=hip_pos[Mapping05[0],1];temp.data[2]:=hip_pos[Mapping05[0],2];
			leg_ref_pos[Mapping05[0]]:= VecAdd( MatMulVec(Rb_target1, VecAdd(temp,MatMulVec(Rleg[Mapping05[0]],BlegCenter_BPosWrtHip[0]))),body_ref_pos);	
		ELSE				
			IsLeg0Move:=FALSE;
			IsLeg5Move:=TRUE;
			EnterLeg5MoveCount:=gait_cycle;
			leg_ref_pos_enter:=leg_ref_pos_last;
		END_IF
		
		//force compensator
		tipForceTarget:=tipForceDesireLegF;
		IF (gait_cycle-EnterBlegCenterCount)<=fceLoadTime*gvl.sampleRate THEN
			tr  := UDINT_TO_LREAL(gait_cycle-EnterBlegCenterCount) / gvl.sampleRate / fceLoadTime;
			fbGetPivot(tNow := tr, tTotal := 1.0, pivot => pvt);
			FOR i:=0 TO 5 DO
				FOR j:=0 TO 2 DO
					tipForceDesire[i,j]:=(1-pvt)*tipForceDesireZeros[i,j]+pvt*tipForceTarget[i,j];
				END_FOR
			END_FOR
		ELSIF (gait_cycle-EnterBlegCenterCount)>(BlegCenterRetractTime+BlegCenterExtendTime-fceLoadTime)*gvl.sampleRate AND (gait_cycle-EnterBlegCenterCount)<=(BlegCenterRetractTime+BlegCenterExtendTime)*gvl.sampleRate THEN
			tr  := (UDINT_TO_LREAL(gait_cycle-EnterBlegCenterCount) / gvl.sampleRate -(BlegCenterRetractTime+BlegCenterExtendTime-fceLoadTime))/ fceLoadTime;
			fbGetPivot(tNow := tr, tTotal := 1.0, pivot => pvt);
			FOR i:=0 TO 5 DO
				FOR j:=0 TO 2 DO
					tipForceDesire[i,j]:=(1-pvt)*tipForceTarget[i,j]+pvt*tipForceDesireZeros[i,j];
				END_FOR
			END_FOR	
		END_IF
		
	END_IF
	
	IF IsLeg5Move=TRUE THEN
		IF (gait_cycle-EnterLeg5MoveCount)<=BlegCenterRetractTime*gvl.sampleRate THEN
			tr  := UDINT_TO_LREAL(gait_cycle-EnterLeg5MoveCount) / gvl.sampleRate / BlegCenterRetractTime;
			fbGetPivot(tNow := tr, tTotal := 1.0, pivot => pvt);
			FOR j:=0 TO 2 DO
				BlegCenter_BJntRef[1].data[j]:=(1-pvt)*BlegCenter_BJntStart[1].data[j]+pvt*(BC_BJntRetract[1,j]);
			END_FOR	
			gvl.legCtrl[Mapping05[1]].ForwardKinetics(motorAngles:=BlegCenter_BJntRef[1].data , legIndex:=Mapping05[1] , tipPosition=>BlegCenter_BPosWrtHip[1].data );
			fbRotMat(yaw := body_ref_ang_enter.data[2], pitch := body_ref_ang_enter.data[1],roll := body_ref_ang_enter.data[0], rm =>  Rb_target1 );
			temp.data[0]:=hip_pos[Mapping05[1],0];temp.data[1]:=hip_pos[Mapping05[1],1];temp.data[2]:=hip_pos[Mapping05[1],2];
			leg_ref_pos[Mapping05[1]]:= VecAdd( MatMulVec(Rb_target1, VecAdd(temp,MatMulVec(Rleg[Mapping05[1]],BlegCenter_BPosWrtHip[1]))),body_ref_pos);
		ELSIF (gait_cycle-EnterLeg5MoveCount)<=(BlegCenterRetractTime+BlegCenterExtendTime)*gvl.sampleRate THEN
			tr  := (UDINT_TO_LREAL(gait_cycle-EnterLeg5MoveCount) / gvl.sampleRate -BlegCenterRetractTime)/ BlegCenterExtendTime;
			fbGetPivot(tNow := tr, tTotal := 1.0, pivot => pvt);
			FOR j:=0 TO 2 DO
				BlegCenter_BJntRef[1].data[j]:=(1-pvt)*BC_BJntRetract[1,j]+pvt*(BC_BJntTarget[1,j]);
			END_FOR
			gvl.legCtrl[Mapping05[1]].ForwardKinetics(motorAngles:=BlegCenter_BJntRef[1].data , legIndex:=Mapping05[1] , tipPosition=>BlegCenter_BPosWrtHip[1].data );
			fbRotMat(yaw := body_ref_ang_enter.data[2], pitch := body_ref_ang_enter.data[1],roll := body_ref_ang_enter.data[0], rm =>  Rb_target1 );
			temp.data[0]:=hip_pos[Mapping05[1],0];temp.data[1]:=hip_pos[Mapping05[1],1];temp.data[2]:=hip_pos[Mapping05[1],2];
			leg_ref_pos[Mapping05[1]]:= VecAdd( MatMulVec(Rb_target1, VecAdd(temp,MatMulVec(Rleg[Mapping05[1]],BlegCenter_BPosWrtHip[1]))),body_ref_pos);
		ELSE			
			IsLeg5Move:=FALSE;
			leg_ref_pos_enter:=leg_ref_pos_last;
			BlegCenterFinished:=TRUE;
			tipForceDesire:=tipForceDesireZeros;
			RequireMlegRollA:=TRUE;//**********************************************************************************************
		END_IF
		
		//force compensator
		tipForceTarget:=tipForceDesireLegA;
		IF (gait_cycle-EnterLeg5MoveCount)<=fceLoadTime*gvl.sampleRate THEN
			tr  := UDINT_TO_LREAL(gait_cycle-EnterLeg5MoveCount) / gvl.sampleRate / fceLoadTime;
			fbGetPivot(tNow := tr, tTotal := 1.0, pivot => pvt);
			FOR i:=0 TO 5 DO
				FOR j:=0 TO 2 DO
					tipForceDesire[i,j]:=(1-pvt)*tipForceDesireZeros[i,j]+pvt*tipForceTarget[i,j];
				END_FOR
			END_FOR
		ELSIF (gait_cycle-EnterLeg5MoveCount)>(BlegCenterRetractTime+BlegCenterExtendTime-fceLoadTime)*gvl.sampleRate AND (gait_cycle-EnterLeg5MoveCount)<=(BlegCenterRetractTime+BlegCenterExtendTime)*gvl.sampleRate THEN
			tr  := (UDINT_TO_LREAL(gait_cycle-EnterLeg5MoveCount) / gvl.sampleRate -(BlegCenterRetractTime+BlegCenterExtendTime-fceLoadTime))/ fceLoadTime;
			fbGetPivot(tNow := tr, tTotal := 1.0, pivot => pvt);
			FOR i:=0 TO 5 DO
				FOR j:=0 TO 2 DO
					tipForceDesire[i,j]:=(1-pvt)*tipForceTarget[i,j]+pvt*tipForceDesireZeros[i,j];
				END_FOR
			END_FOR	
		END_IF		
	END_IF
	
END_IF
END_METHOD

METHOD PUBLIC TrjPlanning_BLegPosAdjust : BOOL
VAR_INPUT
END_VAR

VAR
	i: INT;
	
	tipForceDesireLegA:	 ARRAY[0..5,0..2] OF LREAL:=[0,-100,0,
													 0,0,0,
													 0,0,0,
													 0,0,0,
													 0,0,0,
													 0,0,0];
	tipForceDesireLegF:	 ARRAY[0..5,0..2] OF LREAL:=[0,0,0,
													 0,0,0,
													 0,0,0,
													 0,0,0,
													 0,0,0,
													 0,-120,0];		
	tr: LREAL;
	j: INT;
END_VAR
IF BLegPosAdjustFinished=FALSE THEN
	IF (gait_cycle-EnterBLegPosAdjustCount)<=LREAL_TO_UDINT(BLPA_time)*gvl.sampleRate THEN
		body_ref_ang:=body_ref_ang_enter;
		body_ref_pos:=body_ref_pos_enter;
		leg_ref_pos:=leg_ref_pos_enter;
		i:=0;
		fbElipseInterpolation(x0:=leg_ref_pos_enter[Mapping05[i]].data[0] , y0:=leg_ref_pos_enter[Mapping05[i]].data[1] , z0:=leg_ref_pos_enter[Mapping05[i]].data[2] , x1:=BLPA_tgtLegPos[Mapping05[i]].data[0] , 
		y1:=BLPA_tgtLegPos[Mapping05[i]].data[1] , z1:=BLPA_tgtLegPos[Mapping05[i]].data[2] , h:=BLPA_height , T:=BLPA_time , t0:=0 , tNow:= (gait_cycle-EnterBLegPosAdjustCount)*delta_t, 
		x=>leg_ref_pos[Mapping05[i]].data[0] , y=>leg_ref_pos[Mapping05[i]].data[1] , z=>leg_ref_pos[Mapping05[i]].data[2] );
		IF (gait_cycle-EnterBLegPosAdjustCount)=LREAL_TO_UDINT(BLPA_time)*gvl.sampleRate THEN
			leg_ref_pos_enter_next:=leg_ref_pos;
		END_IF
		
		//force compensator
		tipForceTarget:=tipForceDesireLegF;
		IF (gait_cycle-EnterBLegPosAdjustCount)<=fceLoadTime*gvl.sampleRate THEN
			tr  := UDINT_TO_LREAL(gait_cycle-EnterBLegPosAdjustCount) / gvl.sampleRate / fceLoadTime;
			fbGetPivot(tNow := tr, tTotal := 1.0, pivot => pvt);
			FOR i:=0 TO 5 DO
				FOR j:=0 TO 2 DO
					tipForceDesire[i,j]:=(1-pvt)*tipForceDesireZeros[i,j]+pvt*tipForceTarget[i,j];
				END_FOR
			END_FOR
		ELSIF (gait_cycle-EnterBLegPosAdjustCount)>LREAL_TO_UDINT((BLPA_time-fceLoadTime)*gvl.sampleRate) THEN
			tr  := (UDINT_TO_LREAL(gait_cycle-EnterBLegPosAdjustCount) / gvl.sampleRate -(BLPA_time-fceLoadTime))/ fceLoadTime;
			fbGetPivot(tNow := tr, tTotal := 1.0, pivot => pvt);
			FOR i:=0 TO 5 DO
				FOR j:=0 TO 2 DO
					tipForceDesire[i,j]:=(1-pvt)*tipForceTarget[i,j]+pvt*tipForceDesireZeros[i,j];
				END_FOR
			END_FOR	
		END_IF
		
	ELSIF (gait_cycle-EnterBLegPosAdjustCount)<=LREAL_TO_UDINT(2*BLPA_time)*gvl.sampleRate THEN
		body_ref_ang:=body_ref_ang_enter;
		body_ref_pos:=body_ref_pos_enter;
		leg_ref_pos:=leg_ref_pos_enter_next;
		i:=1;
		fbElipseInterpolation(x0:=leg_ref_pos_enter[Mapping05[i]].data[0] , y0:=leg_ref_pos_enter[Mapping05[i]].data[1] , z0:=leg_ref_pos_enter[Mapping05[i]].data[2] , x1:=BLPA_tgtLegPos[Mapping05[i]].data[0] , 
		y1:=BLPA_tgtLegPos[Mapping05[i]].data[1] , z1:=BLPA_tgtLegPos[Mapping05[i]].data[2] , h:=BLPA_height , T:=BLPA_time , t0:=0 , tNow:= (gait_cycle-EnterBLegPosAdjustCount-LREAL_TO_UDINT(BLPA_time)*gvl.sampleRate)*delta_t, 
		x=>leg_ref_pos[Mapping05[i]].data[0] , y=>leg_ref_pos[Mapping05[i]].data[1] , z=>leg_ref_pos[Mapping05[i]].data[2] );		
		
		//force compensator
		tipForceTarget:=tipForceDesireLegA;
		IF (gait_cycle-EnterBLegPosAdjustCount)<=(BLPA_time+fceLoadTime)*gvl.sampleRate THEN
			tr  := (UDINT_TO_LREAL(gait_cycle-EnterBLegPosAdjustCount) / gvl.sampleRate-BLPA_time )/ fceLoadTime;
			fbGetPivot(tNow := tr, tTotal := 1.0, pivot => pvt);
			FOR i:=0 TO 5 DO
				FOR j:=0 TO 2 DO
					tipForceDesire[i,j]:=(1-pvt)*tipForceDesireZeros[i,j]+pvt*tipForceTarget[i,j];
				END_FOR
			END_FOR
		ELSIF (gait_cycle-EnterBLegPosAdjustCount)>LREAL_TO_UDINT((2*BLPA_time-fceLoadTime)*gvl.sampleRate) THEN
			tr  := (UDINT_TO_LREAL(gait_cycle-EnterBLegPosAdjustCount) / gvl.sampleRate -(2*BLPA_time-fceLoadTime))/ fceLoadTime;
			fbGetPivot(tNow := tr, tTotal := 1.0, pivot => pvt);
			FOR i:=0 TO 5 DO
				FOR j:=0 TO 2 DO
					tipForceDesire[i,j]:=(1-pvt)*tipForceTarget[i,j]+pvt*tipForceDesireZeros[i,j];
				END_FOR
			END_FOR	
		END_IF
		
	ELSE
		BLegPosAdjustFinished:=TRUE;	
		tipForceDesire:=tipForceDesireZeros;
	END_IF
END_IF
END_METHOD

METHOD PUBLIC TrjPlanning_BLegRecovery : BOOL
VAR_INPUT
END_VAR
VAR
	BLR_FPosExtractTarget:ARRAY[0..1,0..2] OF LREAL:=[-0.6,-0.1797+0.06,0,
                                                     -0.6,-0.1797+0.06,0];
	BLR_FPosExtendTarget:ARRAY[0..1,0..2] OF LREAL:=[-0.35,-0.1797,0,
                                                     -0.35,-0.1797,0];												 
	i: INT;
	tr: LREAL;
	j: INT;
	Rb_target1: Mat3;
	temp: vec3;
	tempLeg:ARRAY [0..2] OF LREAL;
	tempJnt:ARRAY [0..2] OF LREAL;
	tempRef:ARRAY [0..2] OF LREAL;	
	
	tipForceDesireLegA:	 ARRAY[0..5,0..2] OF LREAL:=[0,-100,0,
													 0,0,0,
													 0,0,0,
													 0,0,0,
													 0,0,0,
													 0,0,0];
	tipForceDesireLegF:	 ARRAY[0..5,0..2] OF LREAL:=[0,0,0,
													 0,0,0,
													 0,0,0,
													 0,0,0,
													 0,0,0,
													 0,-120,0];			
	
	
END_VAR
IF(gait_cycle-EnterBLegRecoveryCount)=1 THEN
	FOR i:=0 TO 1 DO
		tempLeg[0]:=BLR_FPosExtractTarget[i,0];tempLeg[1]:=BLR_FPosExtractTarget[i,1];tempLeg[2]:=BLR_FPosExtractTarget[i,2];
		tempRef[0]:=BLR_FJntStart[i].data[0];tempRef[1]:=BLR_FJntStart[i].data[1];tempRef[2]:=BLR_FJntStart[i].data[2];
		GVL.legCtrl[Mapping05[i]].InverseKinetics(tipPosition:=tempLeg , refPosLast:=tempRef , legIndex:=Mapping05[i] , motorAngles=>tempJnt , isSingular=> );
		BLR_FJntExtractTarget[i,0]:=tempJnt[0];BLR_FJntExtractTarget[i,1]:=tempJnt[1];BLR_FJntExtractTarget[i,2]:=tempJnt[2];	

		tempLeg[0]:=BLR_FPosExtendTarget[i,0];tempLeg[1]:=BLR_FPosExtendTarget[i,1];tempLeg[2]:=BLR_FPosExtendTarget[i,2];
		tempRef[0]:=BLR_FJntStart[i].data[0];tempRef[1]:=BLR_FJntStart[i].data[1];tempRef[2]:=BLR_FJntStart[i].data[2];
		GVL.legCtrl[Mapping05[i]].InverseKinetics(tipPosition:=tempLeg , refPosLast:=tempRef , legIndex:=Mapping05[i] , motorAngles=>tempJnt , isSingular=> );
		BLR_FJntExtendTarget[i,0]:=tempJnt[0];BLR_FJntExtendTarget[i,1]:=tempJnt[1];BLR_FJntExtendTarget[i,2]:=tempJnt[2];	
	END_FOR
END_IF

IF BLegRecoveryFinished=FALSE THEN
	body_ref_pos:=body_ref_pos_enter;
	body_ref_ang:=body_ref_ang_enter;
	leg_ref_pos:=leg_ref_pos_enter;
	IF(gait_cycle-EnterBLegRecoveryCount)<=BLRRetractTime*gvl.sampleRate THEN
		tr  := UDINT_TO_LREAL(gait_cycle - EnterBLegRecoveryCount) / gvl.sampleRate /BLRRetractTime;
		fbGetPivot(tNow := tr, tTotal := 1.0, pivot => pvt);
		i:=0;
		FOR j:=0 TO 2 DO
			BLR_FJntRef[i].data[j]:=(1-pvt)*BLR_FJntStart[i].data[j]+pvt*(BLR_FJntExtractTarget[i,j]);
		END_FOR
		gvl.legCtrl[Mapping05[i]].ForwardKinetics(motorAngles:=BLR_FJntRef[i].data , legIndex:=Mapping05[i] , tipPosition=>BLR_FPosWrtHip[i].data );
		fbRotMat(yaw := body_ref_ang_enter.data[2], pitch := body_ref_ang_enter.data[1],roll := body_ref_ang_enter.data[0], rm =>  Rb_target1 );
		temp.data[0]:=hip_pos[Mapping05[i],0];temp.data[1]:=hip_pos[Mapping05[i],1];temp.data[2]:=hip_pos[Mapping05[i],2];
		leg_ref_pos[Mapping05[i]]:= VecAdd( MatMulVec(Rb_target1, VecAdd(temp,MatMulVec(Rleg[Mapping05[i]],BLR_FPosWrtHip[i]))),body_ref_pos);

//***************force compensator start************************************************************		
		tipForceTarget:=tipForceDesireLegF;
		IF (gait_cycle-EnterBLegRecoveryCount)<=fceLoadTime*gvl.sampleRate THEN
			tr  := UDINT_TO_LREAL(gait_cycle-EnterBLegRecoveryCount) / gvl.sampleRate / fceLoadTime;
			fbGetPivot(tNow := tr, tTotal := 1.0, pivot => pvt);
			FOR i:=0 TO 5 DO
				FOR j:=0 TO 2 DO
					tipForceDesire[i,j]:=(1-pvt)*tipForceDesireZeros[i,j]+pvt*tipForceTarget[i,j];
				END_FOR
			END_FOR
		END_IF
//***************************end*****************************************************************			
		
	ELSIF (gait_cycle-EnterBLegRecoveryCount)<=(BLRRetractTime+BLRExtendTime)*gvl.sampleRate THEN
		tr  := (UDINT_TO_LREAL(gait_cycle - EnterBLegRecoveryCount) / gvl.sampleRate-BLRRetractTime )/BLRExtendTime;
		fbGetPivot(tNow := tr, tTotal := 1.0, pivot => pvt);
		i:=0;
			FOR j:=0 TO 2 DO
			BLR_FJntRef[i].data[j]:=(1-pvt)*BLR_FJntExtractTarget[i,j]+pvt*(BLR_FJntExtendTarget[i,j]);
		END_FOR
		gvl.legCtrl[Mapping05[i]].ForwardKinetics(motorAngles:=BLR_FJntRef[i].data , legIndex:=Mapping05[i] , tipPosition=>BLR_FPosWrtHip[i].data );
		fbRotMat(yaw := body_ref_ang_enter.data[2], pitch := body_ref_ang_enter.data[1],roll := body_ref_ang_enter.data[0], rm =>  Rb_target1 );
		temp.data[0]:=hip_pos[Mapping05[i],0];temp.data[1]:=hip_pos[Mapping05[i],1];temp.data[2]:=hip_pos[Mapping05[i],2];
		leg_ref_pos[Mapping05[i]]:= VecAdd( MatMulVec(Rb_target1, VecAdd(temp,MatMulVec(Rleg[Mapping05[i]],BLR_FPosWrtHip[i]))),body_ref_pos);
		IF (gait_cycle-EnterBLegRecoveryCount)=LREAL_TO_UDINT((BLRRetractTime+BLRExtendTime)*gvl.sampleRate) THEN
			leg_ref_pos_enter:=leg_ref_pos;
		END_IF
		
//***************force compensator start************************************************************	
		tipForceTarget:=tipForceDesireLegF;	
		IF (gait_cycle-EnterBLegRecoveryCount)>LREAL_TO_UDINT((BLRRetractTime+BLRExtendTime-fceLoadTime)*gvl.sampleRate) THEN
			tr  := (UDINT_TO_LREAL(gait_cycle-EnterBLegRecoveryCount) / gvl.sampleRate -(BLRRetractTime+BLRExtendTime-fceLoadTime))/ fceLoadTime;
			fbGetPivot(tNow := tr, tTotal := 1.0, pivot => pvt);
			FOR i:=0 TO 5 DO
				FOR j:=0 TO 2 DO
					tipForceDesire[i,j]:=(1-pvt)*tipForceTarget[i,j]+pvt*tipForceDesireZeros[i,j];
				END_FOR
			END_FOR	
		END_IF	
//*************************end***********************************************************************			
		
	ELSIF (gait_cycle-EnterBLegRecoveryCount)<=(2*BLRRetractTime+BLRExtendTime)*gvl.sampleRate THEN	
		tr  := (UDINT_TO_LREAL(gait_cycle - EnterBLegRecoveryCount) / gvl.sampleRate-BLRRetractTime-BLRExtendTime )/BLRRetractTime;
		fbGetPivot(tNow := tr, tTotal := 1.0, pivot => pvt);
		i:=1;
		FOR j:=0 TO 2 DO
			BLR_FJntRef[i].data[j]:=(1-pvt)*BLR_FJntStart[i].data[j]+pvt*(BLR_FJntExtractTarget[i,j]);
		END_FOR
		gvl.legCtrl[Mapping05[i]].ForwardKinetics(motorAngles:=BLR_FJntRef[i].data , legIndex:=Mapping05[i] , tipPosition=>BLR_FPosWrtHip[i].data );
		fbRotMat(yaw := body_ref_ang_enter.data[2], pitch := body_ref_ang_enter.data[1],roll := body_ref_ang_enter.data[0], rm =>  Rb_target1 );
		temp.data[0]:=hip_pos[Mapping05[i],0];temp.data[1]:=hip_pos[Mapping05[i],1];temp.data[2]:=hip_pos[Mapping05[i],2];
		leg_ref_pos[Mapping05[i]]:= VecAdd( MatMulVec(Rb_target1, VecAdd(temp,MatMulVec(Rleg[Mapping05[i]],BLR_FPosWrtHip[i]))),body_ref_pos);	
		
//***************force compensator start************************************************************		
		tipForceTarget:=tipForceDesireLegA;
		IF (gait_cycle-EnterBLegRecoveryCount)<=(BLRRetractTime+BLRExtendTime+fceLoadTime)*gvl.sampleRate THEN
			tr  := (UDINT_TO_LREAL(gait_cycle-EnterBLegRecoveryCount) / gvl.sampleRate-(BLRRetractTime+BLRExtendTime) )/ fceLoadTime;
			fbGetPivot(tNow := tr, tTotal := 1.0, pivot => pvt);
			FOR i:=0 TO 5 DO
				FOR j:=0 TO 2 DO
					tipForceDesire[i,j]:=(1-pvt)*tipForceDesireZeros[i,j]+pvt*tipForceTarget[i,j];
				END_FOR
			END_FOR
		END_IF
//**************************end******************************************************************				
		
	ELSIF (gait_cycle-EnterBLegRecoveryCount)<=(2*BLRRetractTime+2*BLRExtendTime)*gvl.sampleRate THEN	
		tr  := (UDINT_TO_LREAL(gait_cycle - EnterBLegRecoveryCount) / gvl.sampleRate-2*BLRRetractTime-BLRExtendTime )/BLRExtendTime;
		fbGetPivot(tNow := tr, tTotal := 1.0, pivot => pvt);
		i:=1;
		FOR j:=0 TO 2 DO
			BLR_FJntRef[i].data[j]:=(1-pvt)*BLR_FJntExtractTarget[i,j]+pvt*(BLR_FJntExtendTarget[i,j]);
		END_FOR
		gvl.legCtrl[Mapping05[i]].ForwardKinetics(motorAngles:=BLR_FJntRef[i].data , legIndex:=Mapping05[i] , tipPosition=>BLR_FPosWrtHip[i].data );
		fbRotMat(yaw := body_ref_ang_enter.data[2], pitch := body_ref_ang_enter.data[1],roll := body_ref_ang_enter.data[0], rm =>  Rb_target1 );
		temp.data[0]:=hip_pos[Mapping05[i],0];temp.data[1]:=hip_pos[Mapping05[i],1];temp.data[2]:=hip_pos[Mapping05[i],2];
		leg_ref_pos[Mapping05[i]]:= VecAdd( MatMulVec(Rb_target1, VecAdd(temp,MatMulVec(Rleg[Mapping05[i]],BLR_FPosWrtHip[i]))),body_ref_pos);
		IF 	(gait_cycle-EnterBLegRecoveryCount)=LREAL_TO_UDINT((2*BLRRetractTime+2*BLRExtendTime)*gvl.sampleRate) THEN
			leg_ref_pos_enter:=leg_ref_pos;
		END_IF	
		
//***************force compensator start************************************************************	
		tipForceTarget:=tipForceDesireLegA;	
		IF (gait_cycle-EnterBLegRecoveryCount)>LREAL_TO_UDINT((2*BLRRetractTime+2*BLRExtendTime-fceLoadTime)*gvl.sampleRate) THEN
			tr  := (UDINT_TO_LREAL(gait_cycle-EnterBLegRecoveryCount) / gvl.sampleRate -(2*BLRRetractTime+2*BLRExtendTime-fceLoadTime))/ fceLoadTime;
			fbGetPivot(tNow := tr, tTotal := 1.0, pivot => pvt);
			FOR i:=0 TO 5 DO
				FOR j:=0 TO 2 DO
					tipForceDesire[i,j]:=(1-pvt)*tipForceTarget[i,j]+pvt*tipForceDesireZeros[i,j];
				END_FOR
			END_FOR	
		END_IF	
//**********************end**********************************************************************		
		
	ELSE	
		body_ref_pos_enter:=body_ref_pos;
		body_ref_ang_enter:=body_ref_ang;
		leg_ref_pos_enter:=leg_ref_pos;
		BLegRecoveryFinished:=TRUE;
		tipForceDesire:=tipForceDesireZeros;
		RequireMlegRollC:=TRUE;
	END_IF
END_IF
END_METHOD

METHOD PUBLIC TrjPlanning_BodyPosAdjust : BOOL
VAR_INPUT
END_VAR

VAR
	tr: LREAL;
	i: INT;
	Rb_target1: Mat3;
	temp: VEC3;
	j: INT;
	
	tipForceDesireLegA:	 ARRAY[0..5,0..2] OF LREAL:=[0,-200,0,
													 0,0,0,
													 0,0,0,
													 0,0,0,
													 0,0,0,
													 0,0,0];
	tipForceDesireLegF:	 ARRAY[0..5,0..2] OF LREAL:=[0,0,0,
													 0,0,0,
													 0,0,0,
													 0,0,0,
													 0,0,0,
													 0,-220,0];			
END_VAR
IF BodyPosAdjustFinished=FALSE AND (gait_cycle-EnterBodyPosAdjustCount)<=LREAL_TO_UDINT((2*BPA_LiftGroundTime+BPA_AdjustTime+3*BPA_AdjustExtractTime+3*BPA_AdjustExtendTime)*gvl.sampleRate) THEN
	IF (gait_cycle-EnterBodyPosAdjustCount)<=LREAL_TO_UDINT((BPA_LiftGroundTime)*gvl.sampleRate) THEN
		leg_ref_pos:=leg_ref_pos_enter;
		body_ref_ang:=BPA_BodyAngStart;
		body_ref_pos:=BPA_BodyPosStart;
		tr  := UDINT_TO_LREAL(gait_cycle - EnterBodyPosAdjustCount) / gvl.sampleRate /BPA_LiftGroundTime;
		fbGetPivot(tNow := tr, tTotal := 1.0, pivot => pvt);	
		body_ref_pos.data[2]:=(1-pvt)*BPA_BodyPosStart.data[2]+pvt*(BPA_BodyPosStart.data[2]+BPA_HeightAdd);
		FOR i:=0 TO 1 DO
			gvl.legCtrl[Mapping23[i]].ForwardKinetics(motorAngles:=BPA_FJntRef[i].data , legIndex:=Mapping23[i] , tipPosition=>BPA_FPosWrtHip[i].data );
			fbRotMat(yaw := body_ref_ang.data[2], pitch := body_ref_ang.data[1],roll := body_ref_ang.data[0], rm =>  Rb_target1 );
			temp.data[0]:=hip_pos[Mapping23[i],0];temp.data[1]:=hip_pos[Mapping23[i],1];temp.data[2]:=hip_pos[Mapping23[i],2];
			leg_ref_pos[Mapping23[i]]:= VecAdd( MatMulVec(Rb_target1, VecAdd(temp,MatMulVec(Rleg[Mapping23[i]],BPA_FPosWrtHip[i]))),body_ref_pos);			
		END_FOR
	ELSIF (gait_cycle-EnterBodyPosAdjustCount)<=LREAL_TO_UDINT((BPA_LiftGroundTime+BPA_AdjustTime)*gvl.sampleRate) THEN	
		leg_ref_pos:=leg_ref_pos_enter;
		tr  := (UDINT_TO_LREAL(gait_cycle - EnterBodyPosAdjustCount) / gvl.sampleRate -BPA_LiftGroundTime)/BPA_AdjustTime;
		fbGetPivot(tNow := tr, tTotal := 1.0, pivot => pvt);		
		FOR i:=0 TO 2 DO
			body_ref_pos.data[i]:=(1-pvt)*BPA_BodyPosStart.data[i]+pvt*BPA_BodyPoseEnd.data[i];
			body_ref_ang.data[i]:=(1-pvt)*BPA_BodyAngStart.data[i]+pvt*BPA_BodyAngEnd.data[i];
		END_FOR	
		body_ref_pos.data[2]:=body_ref_pos.data[2]+BPA_HeightAdd;
		FOR i:=0 TO 1 DO
			gvl.legCtrl[Mapping23[i]].ForwardKinetics(motorAngles:=BPA_FJntRef[i].data , legIndex:=Mapping23[i] , tipPosition=>BPA_FPosWrtHip[i].data );
			fbRotMat(yaw := body_ref_ang.data[2], pitch := body_ref_ang.data[1],roll := body_ref_ang.data[0], rm =>  Rb_target1 );
			temp.data[0]:=hip_pos[Mapping23[i],0];temp.data[1]:=hip_pos[Mapping23[i],1];temp.data[2]:=hip_pos[Mapping23[i],2];
			leg_ref_pos[Mapping23[i]]:= VecAdd( MatMulVec(Rb_target1, VecAdd(temp,MatMulVec(Rleg[Mapping23[i]],BPA_FPosWrtHip[i]))),body_ref_pos);						
		END_FOR
	ELSIF (gait_cycle-EnterBodyPosAdjustCount)<=LREAL_TO_UDINT((2*BPA_LiftGroundTime+BPA_AdjustTime)*gvl.sampleRate) THEN		
		leg_ref_pos:=leg_ref_pos_enter;
		body_ref_ang:=BPA_BodyAngEnd;
		body_ref_pos:=BPA_BodyPoseEnd;	
		tr  := (UDINT_TO_LREAL(gait_cycle - EnterBodyPosAdjustCount) / gvl.sampleRate-BPA_LiftGroundTime-BPA_AdjustTime )/BPA_LiftGroundTime;
		fbGetPivot(tNow := tr, tTotal := 1.0, pivot => pvt);		
		body_ref_pos.data[2]:=(1-pvt)*(BPA_BodyPosStart.data[2]+BPA_HeightAdd)+pvt*BPA_BodyPosStart.data[2];
		FOR i:=0 TO 1 DO
			gvl.legCtrl[Mapping23[i]].ForwardKinetics(motorAngles:=BPA_FJntRef[i].data , legIndex:=Mapping23[i] , tipPosition=>BPA_FPosWrtHip[i].data );
			fbRotMat(yaw := body_ref_ang.data[2], pitch := body_ref_ang.data[1],roll := body_ref_ang.data[0], rm =>  Rb_target1 );
			temp.data[0]:=hip_pos[Mapping23[i],0];temp.data[1]:=hip_pos[Mapping23[i],1];temp.data[2]:=hip_pos[Mapping23[i],2];
			leg_ref_pos[Mapping23[i]]:= VecAdd( MatMulVec(Rb_target1, VecAdd(temp,MatMulVec(Rleg[Mapping23[i]],BPA_FPosWrtHip[i]))),body_ref_pos);				
		END_FOR
		IF (gait_cycle-EnterBodyPosAdjustCount)=LREAL_TO_UDINT((2*BPA_LiftGroundTime+BPA_AdjustTime)*gvl.sampleRate) THEN
			BPA_legPosEnterExtract:=leg_ref_pos;
			FOR i:=0 TO 1 DO
				FOR j:=0 TO 2 DO
					BPA_MJntStart[i].data[j]:=jointPosLast[Mapping14[i],j];
					BPA_BJntStart[i].data[j]:=jointPosLast[Mapping05[i],j];
				END_FOR
			END_FOR			
		END_IF
	ELSIF (gait_cycle-EnterBodyPosAdjustCount)<=LREAL_TO_UDINT((2*BPA_LiftGroundTime+BPA_AdjustTime+BPA_AdjustExtractTime)*gvl.sampleRate) THEN		
		body_ref_pos:=BPA_BodyPoseEnd;
		body_ref_ang:=BPA_BodyAngEnd;
		leg_ref_pos:=BPA_legPosEnterExtract;
		tr  := (UDINT_TO_LREAL(gait_cycle - EnterBodyPosAdjustCount) / gvl.sampleRate-2*BPA_LiftGroundTime-BPA_AdjustTime )/BPA_AdjustExtractTime;
		fbGetPivot(tNow := tr, tTotal := 1.0, pivot => pvt);
		FOR i:=0 TO 1 DO
			FOR j:=0 TO 2 DO
				BPA_MJntRef[i].data[j]:=(1-pvt)*BPA_MJntStart[i].data[j]+pvt*BPA_MJntExtract[i,j];
			END_FOR			
			gvl.legCtrl[Mapping14[i]].ForwardKinetics(motorAngles:=BPA_MJntRef[i].data , legIndex:=Mapping14[i] , tipPosition=>BPA_MPosWrtHip[i].data );
			fbRotMat(yaw := body_ref_ang.data[2], pitch := body_ref_ang.data[1],roll := body_ref_ang.data[0], rm =>  Rb_target1 );
			temp.data[0]:=hip_pos[Mapping14[i],0];temp.data[1]:=hip_pos[Mapping14[i],1];temp.data[2]:=hip_pos[Mapping14[i],2];
			leg_ref_pos[Mapping14[i]]:= VecAdd( MatMulVec(Rb_target1, VecAdd(temp,MatMulVec(Rleg[Mapping14[i]],BPA_MPosWrtHip[i]))),body_ref_pos);

			gvl.legCtrl[Mapping23[i]].ForwardKinetics(motorAngles:=BPA_FJntRef[i].data , legIndex:=Mapping23[i] , tipPosition=>BPA_FPosWrtHip[i].data );
			temp.data[0]:=hip_pos[Mapping23[i],0];temp.data[1]:=hip_pos[Mapping23[i],1];temp.data[2]:=hip_pos[Mapping23[i],2];
			leg_ref_pos[Mapping23[i]]:= VecAdd( MatMulVec(Rb_target1, VecAdd(temp,MatMulVec(Rleg[Mapping23[i]],BPA_FPosWrtHip[i]))),body_ref_pos);	
		END_FOR
	ELSIF (gait_cycle-EnterBodyPosAdjustCount)<=LREAL_TO_UDINT((2*BPA_LiftGroundTime+BPA_AdjustTime+BPA_AdjustExtractTime+BPA_AdjustExtendTime)*gvl.sampleRate) THEN	
		body_ref_pos:=BPA_BodyPoseEnd;
		body_ref_ang:=BPA_BodyAngEnd;
		leg_ref_pos:=BPA_legPosEnterExtract;
		tr  := (UDINT_TO_LREAL(gait_cycle - EnterBodyPosAdjustCount) / gvl.sampleRate-2*BPA_LiftGroundTime-BPA_AdjustTime-BPA_AdjustExtractTime )/BPA_AdjustExtendTime;
		fbGetPivot(tNow := tr, tTotal := 1.0, pivot => pvt);	
		FOR i:=0 TO 1 DO
			FOR j:=0 TO 2 DO
				BPA_MJntRef[i].data[j]:=(1-pvt)*BPA_MJntExtract[i,j]+pvt*BPA_MJntExtend[i,j];
			END_FOR
			gvl.legCtrl[Mapping14[i]].ForwardKinetics(motorAngles:=BPA_MJntRef[i].data , legIndex:=Mapping14[i] , tipPosition=>BPA_MPosWrtHip[i].data );
			fbRotMat(yaw := body_ref_ang.data[2], pitch := body_ref_ang.data[1],roll := body_ref_ang.data[0], rm =>  Rb_target1 );
			temp.data[0]:=hip_pos[Mapping14[i],0];temp.data[1]:=hip_pos[Mapping14[i],1];temp.data[2]:=hip_pos[Mapping14[i],2];
			leg_ref_pos[Mapping14[i]]:= VecAdd( MatMulVec(Rb_target1, VecAdd(temp,MatMulVec(Rleg[Mapping14[i]],BPA_MPosWrtHip[i]))),body_ref_pos);
			
			gvl.legCtrl[Mapping23[i]].ForwardKinetics(motorAngles:=BPA_FJntRef[i].data , legIndex:=Mapping23[i] , tipPosition=>BPA_FPosWrtHip[i].data );
			temp.data[0]:=hip_pos[Mapping23[i],0];temp.data[1]:=hip_pos[Mapping23[i],1];temp.data[2]:=hip_pos[Mapping23[i],2];
			leg_ref_pos[Mapping23[i]]:= VecAdd( MatMulVec(Rb_target1, VecAdd(temp,MatMulVec(Rleg[Mapping23[i]],BPA_FPosWrtHip[i]))),body_ref_pos);		
		END_FOR
		IF (gait_cycle-EnterBodyPosAdjustCount)=LREAL_TO_UDINT((2*BPA_LiftGroundTime+BPA_AdjustTime+BPA_AdjustExtractTime+BPA_AdjustExtendTime)*gvl.sampleRate) THEN
			BPA_legPosEnterExtract:=leg_ref_pos;
			FOR i:=0 TO 1 DO
				FOR j:=0 TO 2 DO
					BPA_BJntStart[i].data[j]:=jointPosLast[Mapping05[i],j];
				END_FOR
			END_FOR			
		END_IF
	ELSIF (gait_cycle-EnterBodyPosAdjustCount)<=LREAL_TO_UDINT((2*BPA_LiftGroundTime+BPA_AdjustTime+2*BPA_AdjustExtractTime+BPA_AdjustExtendTime)*gvl.sampleRate) THEN	
		body_ref_pos:=BPA_BodyPoseEnd;
		body_ref_ang:=BPA_BodyAngEnd;
		leg_ref_pos:=BPA_legPosEnterExtract;
		tr  := (UDINT_TO_LREAL(gait_cycle - EnterBodyPosAdjustCount) / gvl.sampleRate-2*BPA_LiftGroundTime-BPA_AdjustTime-BPA_AdjustExtractTime-BPA_AdjustExtendTime )/BPA_AdjustExtractTime;
		fbGetPivot(tNow := tr, tTotal := 1.0, pivot => pvt);
		i:=0;
		FOR j:=0 TO 2 DO
			BPA_BJntRef[i].data[j]:=(1-pvt)*BPA_BJntStart[i].data[j]+pvt*BPA_BJntExtract[i,j];
		END_FOR	
		gvl.legCtrl[Mapping05[i]].ForwardKinetics(motorAngles:=BPA_BJntRef[i].data , legIndex:=Mapping05[i] , tipPosition=>BPA_BPosWrtHip[i].data );
		fbRotMat(yaw := body_ref_ang.data[2], pitch := body_ref_ang.data[1],roll := body_ref_ang.data[0], rm =>  Rb_target1 );
		temp.data[0]:=hip_pos[Mapping05[i],0];temp.data[1]:=hip_pos[Mapping05[i],1];temp.data[2]:=hip_pos[Mapping05[i],2];
		leg_ref_pos[Mapping05[i]]:= VecAdd( MatMulVec(Rb_target1, VecAdd(temp,MatMulVec(Rleg[Mapping05[i]],BPA_BPosWrtHip[i]))),body_ref_pos);
		IF (gait_cycle-EnterBodyPosAdjustCount)=LREAL_TO_UDINT((2*BPA_LiftGroundTime+BPA_AdjustTime+2*BPA_AdjustExtractTime+BPA_AdjustExtendTime)*gvl.sampleRate) THEN
			BPA_legPosEnterExtract:=leg_ref_pos;
			FOR i:=0 TO 1 DO
				FOR j:=0 TO 2 DO
					BPA_BJntStart[i].data[j]:=jointPosLast[Mapping05[i],j];
				END_FOR
			END_FOR			
		END_IF
		
		//force compensator
		tipForceTarget:=tipForceDesireLegF;
		IF (gait_cycle-EnterBodyPosAdjustCount)<=LREAL_TO_UDINT((2*BPA_LiftGroundTime+BPA_AdjustTime+BPA_AdjustExtractTime+BPA_AdjustExtendTime+fceLoadTime)*gvl.sampleRate) THEN
			tr  := (UDINT_TO_LREAL(gait_cycle-EnterBodyPosAdjustCount) / gvl.sampleRate-(2*BPA_LiftGroundTime+BPA_AdjustTime+BPA_AdjustExtractTime+BPA_AdjustExtendTime) )/ fceLoadTime;
			fbGetPivot(tNow := tr, tTotal := 1.0, pivot => pvt);
			FOR i:=0 TO 5 DO
				FOR j:=0 TO 2 DO
					tipForceDesire[i,j]:=(1-pvt)*tipForceDesireZeros[i,j]+pvt*tipForceTarget[i,j];
				END_FOR
			END_FOR
		END_IF

	ELSIF (gait_cycle-EnterBodyPosAdjustCount)<=LREAL_TO_UDINT((2*BPA_LiftGroundTime+BPA_AdjustTime+2*BPA_AdjustExtractTime+2*BPA_AdjustExtendTime)*gvl.sampleRate) THEN	 					
		body_ref_pos:=BPA_BodyPoseEnd;
		body_ref_ang:=BPA_BodyAngEnd;
		leg_ref_pos:=BPA_legPosEnterExtract;					
		tr  := (UDINT_TO_LREAL(gait_cycle - EnterBodyPosAdjustCount) / gvl.sampleRate-2*BPA_LiftGroundTime-BPA_AdjustTime-2*BPA_AdjustExtractTime-BPA_AdjustExtendTime )/BPA_AdjustExtendTime;
		fbGetPivot(tNow := tr, tTotal := 1.0, pivot => pvt);		
		i:=0; 
		FOR j:=0 TO 2 DO
			BPA_BJntRef[i].data[j]:=(1-pvt)*BPA_BJntExtract[i,j]+pvt*BPA_BJntExtend[i,j];
		END_FOR
		gvl.legCtrl[Mapping05[i]].ForwardKinetics(motorAngles:=BPA_BJntRef[i].data , legIndex:=Mapping05[i] , tipPosition=>BPA_BPosWrtHip[i].data );
		fbRotMat(yaw := body_ref_ang.data[2], pitch := body_ref_ang.data[1],roll := body_ref_ang.data[0], rm =>  Rb_target1 );
		temp.data[0]:=hip_pos[Mapping05[i],0];temp.data[1]:=hip_pos[Mapping05[i],1];temp.data[2]:=hip_pos[Mapping05[i],2];
		leg_ref_pos[Mapping05[i]]:= VecAdd( MatMulVec(Rb_target1, VecAdd(temp,MatMulVec(Rleg[Mapping05[i]],BPA_BPosWrtHip[i]))),body_ref_pos);	
		IF (gait_cycle-EnterBodyPosAdjustCount)=LREAL_TO_UDINT((2*BPA_LiftGroundTime+BPA_AdjustTime+2*BPA_AdjustExtractTime+2*BPA_AdjustExtendTime)*gvl.sampleRate) THEN
			BPA_legPosEnterExtract:=leg_ref_pos;
			FOR i:=0 TO 1 DO
				FOR j:=0 TO 2 DO
					BPA_BJntStart[i].data[j]:=jointPosLast[Mapping05[i],j];
				END_FOR
			END_FOR			
		END_IF
		
		//force compensator
		tipForceTarget:=tipForceDesireLegF;
		IF (gait_cycle-EnterBodyPosAdjustCount)>LREAL_TO_UDINT((2*BPA_LiftGroundTime+BPA_AdjustTime+2*BPA_AdjustExtractTime+2*BPA_AdjustExtendTime-fceLoadTime)*gvl.sampleRate)THEN
			tr  := (UDINT_TO_LREAL(gait_cycle-EnterBodyPosAdjustCount) / gvl.sampleRate-(2*BPA_LiftGroundTime+BPA_AdjustTime+2*BPA_AdjustExtractTime+2*BPA_AdjustExtendTime-fceLoadTime) )/ fceLoadTime;
			fbGetPivot(tNow := tr, tTotal := 1.0, pivot => pvt);
			FOR i:=0 TO 5 DO
				FOR j:=0 TO 2 DO
					tipForceDesire[i,j]:=(1-pvt)*tipForceTarget[i,j]+pvt*tipForceDesireZeros[i,j];
				END_FOR
			END_FOR
		END_IF
		
	ELSIF (gait_cycle-EnterBodyPosAdjustCount)<=LREAL_TO_UDINT((2*BPA_LiftGroundTime+BPA_AdjustTime+3*BPA_AdjustExtractTime+2*BPA_AdjustExtendTime)*gvl.sampleRate) THEN
		body_ref_pos:=BPA_BodyPoseEnd;
		body_ref_ang:=BPA_BodyAngEnd;
		leg_ref_pos:=BPA_legPosEnterExtract;
		tr  := (UDINT_TO_LREAL(gait_cycle - EnterBodyPosAdjustCount) / gvl.sampleRate-2*BPA_LiftGroundTime-BPA_AdjustTime-2*BPA_AdjustExtractTime-2*BPA_AdjustExtendTime )/BPA_AdjustExtractTime;
		fbGetPivot(tNow := tr, tTotal := 1.0, pivot => pvt);
		i:=1;
		FOR j:=0 TO 2 DO
			BPA_BJntRef[i].data[j]:=(1-pvt)*BPA_BJntStart[i].data[j]+pvt*BPA_BJntExtract[i,j];
		END_FOR	
		gvl.legCtrl[Mapping05[i]].ForwardKinetics(motorAngles:=BPA_BJntRef[i].data , legIndex:=Mapping05[i] , tipPosition=>BPA_BPosWrtHip[i].data );
		fbRotMat(yaw := body_ref_ang.data[2], pitch := body_ref_ang.data[1],roll := body_ref_ang.data[0], rm =>  Rb_target1 );
		temp.data[0]:=hip_pos[Mapping05[i],0];temp.data[1]:=hip_pos[Mapping05[i],1];temp.data[2]:=hip_pos[Mapping05[i],2];
		leg_ref_pos[Mapping05[i]]:= VecAdd( MatMulVec(Rb_target1, VecAdd(temp,MatMulVec(Rleg[Mapping05[i]],BPA_BPosWrtHip[i]))),body_ref_pos);
		IF (gait_cycle-EnterBodyPosAdjustCount)=LREAL_TO_UDINT((2*BPA_LiftGroundTime+BPA_AdjustTime+3*BPA_AdjustExtractTime+2*BPA_AdjustExtendTime)*gvl.sampleRate) THEN
			BPA_legPosEnterExtract:=leg_ref_pos;
			FOR i:=0 TO 1 DO
				FOR j:=0 TO 2 DO
					BPA_BJntStart[i].data[j]:=jointPosLast[Mapping05[i],j];
				END_FOR
			END_FOR			
		END_IF	
		
		//force compensator
		tipForceTarget:=tipForceDesireLegA;
		IF (gait_cycle-EnterBodyPosAdjustCount)<=LREAL_TO_UDINT((2*BPA_LiftGroundTime+BPA_AdjustTime+2*BPA_AdjustExtractTime+2*BPA_AdjustExtendTime)*gvl.sampleRate) THEN
			tr  := (UDINT_TO_LREAL(gait_cycle-EnterBodyPosAdjustCount) / gvl.sampleRate-(2*BPA_LiftGroundTime+BPA_AdjustTime+BPA_AdjustExtractTime+BPA_AdjustExtendTime+fceLoadTime) )/ fceLoadTime;
			fbGetPivot(tNow := tr, tTotal := 1.0, pivot => pvt);
			FOR i:=0 TO 5 DO
				FOR j:=0 TO 2 DO
					tipForceDesire[i,j]:=(1-pvt)*tipForceDesireZeros[i,j]+pvt*tipForceTarget[i,j];
				END_FOR
			END_FOR
		END_IF
		
	ELSE
		body_ref_pos:=BPA_BodyPoseEnd;
		body_ref_ang:=BPA_BodyAngEnd;
		leg_ref_pos:=BPA_legPosEnterExtract;					
		tr  := (UDINT_TO_LREAL(gait_cycle - EnterBodyPosAdjustCount) / gvl.sampleRate-2*BPA_LiftGroundTime-BPA_AdjustTime-3*BPA_AdjustExtractTime-2*BPA_AdjustExtendTime )/BPA_AdjustExtendTime;
		fbGetPivot(tNow := tr, tTotal := 1.0, pivot => pvt);		
		i:=1; 
		FOR j:=0 TO 2 DO
			BPA_BJntRef[i].data[j]:=(1-pvt)*BPA_BJntExtract[i,j]+pvt*BPA_BJntExtend[i,j];
		END_FOR
		gvl.legCtrl[Mapping05[i]].ForwardKinetics(motorAngles:=BPA_BJntRef[i].data , legIndex:=Mapping05[i] , tipPosition=>BPA_BPosWrtHip[i].data );
		fbRotMat(yaw := body_ref_ang.data[2], pitch := body_ref_ang.data[1],roll := body_ref_ang.data[0], rm =>  Rb_target1 );
		temp.data[0]:=hip_pos[Mapping05[i],0];temp.data[1]:=hip_pos[Mapping05[i],1];temp.data[2]:=hip_pos[Mapping05[i],2];
		leg_ref_pos[Mapping05[i]]:= VecAdd( MatMulVec(Rb_target1, VecAdd(temp,MatMulVec(Rleg[Mapping05[i]],BPA_BPosWrtHip[i]))),body_ref_pos);	
		
		//force compensator
		tipForceTarget:=tipForceDesireLegA;
		IF (gait_cycle-EnterBodyPosAdjustCount)>LREAL_TO_UDINT((2*BPA_LiftGroundTime+BPA_AdjustTime+3*BPA_AdjustExtractTime+3*BPA_AdjustExtendTime-fceLoadTime)*gvl.sampleRate) THEN
			tr  := (UDINT_TO_LREAL(gait_cycle-EnterBodyPosAdjustCount) / gvl.sampleRate-(2*BPA_LiftGroundTime+BPA_AdjustTime+3*BPA_AdjustExtractTime+3*BPA_AdjustExtendTime-fceLoadTime) )/ fceLoadTime;
			fbGetPivot(tNow := tr, tTotal := 1.0, pivot => pvt);
			FOR i:=0 TO 5 DO
				FOR j:=0 TO 2 DO
					tipForceDesire[i,j]:=(1-pvt)*tipForceTarget[i,j]+pvt*tipForceDesireZeros[i,j];
				END_FOR
			END_FOR
		END_IF
		
	END_IF
ELSE
	BodyPosAdjustFinished:=TRUE;
	tipForceDesire:=tipForceDesireZeros;
END_IF
END_METHOD

METHOD PUBLIC TrjPlanning_FlegRotA : BOOL
VAR_INPUT
END_VAR
VAR
	FlegRotA_FJntState1:ARRAY[0..1,0..2] OF LREAL:=[0*pi/180,(162+1)*pi/180,81.588*pi/180,
                                                    0*pi/180,(162+1)*pi/180,81.588*pi/180];	//thigh rotates to grip position
	FlegRotA_FJntState2:ARRAY[0..1,0..2] OF LREAL:=[0*pi/180,(162+1)*pi/180,172*pi/180,
                                                    0*pi/180,(162+1)*pi/180,172*pi/180];	//shank rotates to 	grip position													
	FlegRotA_FJntState3:ARRAY[0..1,0..2] OF LREAL:=[-90*pi/180,(162+1)*pi/180,172*pi/180,
                                                    90*pi/180,(162+1)*pi/180,172*pi/180];	//side rotates to grip position										 
	State1Time:LREAL:=1;
	State2Time:LREAL:=1;
	State3Time:LREAL:=1;
	State4Time:LREAL:=1;
										 
	tr: LREAL;
	i: INT;
	j: INT;
	Rb_target1: Mat3;
	temp: vec3;
	
END_VAR
IF FlegRotAFinished=FALSE THEN
	IF(gait_cycle-EnterFlegRotACount)<=State1Time*gvl.sampleRate THEN
		body_ref_pos:=body_ref_pos_enter;
		body_ref_ang:=body_ref_ang_enter;
		leg_ref_pos:=leg_ref_pos_enter;	
		
		tr  := UDINT_TO_LREAL(gait_cycle - EnterFlegRotACount) / gvl.sampleRate / State1Time;
		fbGetPivot(tNow := tr, tTotal := 1.0, pivot => pvt);	
		FOR i:=0 TO 1 DO
			FOR j:=0 TO 2 DO
				FlegRotA_FJntRef[i].data[j]:=(1-pvt)*FlegRotA_FJntStart[i].data[j]+pvt*(FlegRotA_FJntState1[i,j]);
			END_FOR
			gvl.legCtrl[Mapping23[i]].ForwardKinetics(motorAngles:=FlegRotA_FJntRef[i].data , legIndex:=Mapping23[i] , tipPosition=>FlegRotA_FPosWrtHip[i].data );
			fbRotMat(yaw := body_ref_ang_enter.data[2], pitch := body_ref_ang_enter.data[1],roll := body_ref_ang_enter.data[0], rm =>  Rb_target1 );
			temp.data[0]:=hip_pos[Mapping23[i],0];temp.data[1]:=hip_pos[Mapping23[i],1];temp.data[2]:=hip_pos[Mapping23[i],2];
			leg_ref_pos[Mapping23[i]]:= VecAdd( MatMulVec(Rb_target1, VecAdd(temp,MatMulVec(Rleg[Mapping23[i]],FlegRotA_FPosWrtHip[i]))),body_ref_pos);	
		END_FOR
		
	ELSIF (gait_cycle-EnterFlegRotACount)<=(State1Time+State2Time)*gvl.sampleRate THEN
		body_ref_pos:=body_ref_pos_enter;
		body_ref_ang:=body_ref_ang_enter;
		leg_ref_pos:=leg_ref_pos_enter;	
		
		tr  := (UDINT_TO_LREAL(gait_cycle - EnterFlegRotACount) / gvl.sampleRate-State1Time) / State2Time;
		fbGetPivot(tNow := tr, tTotal := 1.0, pivot => pvt);	
		FOR i:=0 TO 1 DO
			FOR j:=0 TO 2 DO
				FlegRotA_FJntRef[i].data[j]:=(1-pvt)*FlegRotA_FJntState1[i,j]+pvt*(FlegRotA_FJntState2[i,j]);
			END_FOR
			gvl.legCtrl[Mapping23[i]].ForwardKinetics(motorAngles:=FlegRotA_FJntRef[i].data , legIndex:=Mapping23[i] , tipPosition=>FlegRotA_FPosWrtHip[i].data );
			fbRotMat(yaw := body_ref_ang_enter.data[2], pitch := body_ref_ang_enter.data[1],roll := body_ref_ang_enter.data[0], rm =>  Rb_target1 );
			temp.data[0]:=hip_pos[Mapping23[i],0];temp.data[1]:=hip_pos[Mapping23[i],1];temp.data[2]:=hip_pos[Mapping23[i],2];
			leg_ref_pos[Mapping23[i]]:= VecAdd( MatMulVec(Rb_target1, VecAdd(temp,MatMulVec(Rleg[Mapping23[i]],FlegRotA_FPosWrtHip[i]))),body_ref_pos);	
		END_FOR	
	ELSIF	(gait_cycle-EnterFlegRotACount)<=(State1Time+State2Time+State3Time)*gvl.sampleRate THEN
		body_ref_pos:=body_ref_pos_enter;
		body_ref_ang:=body_ref_ang_enter;
		leg_ref_pos:=leg_ref_pos_enter;	
		tr  := (UDINT_TO_LREAL(gait_cycle - EnterFlegRotACount) / gvl.sampleRate-State1Time-State2Time) / State3Time;
		fbGetPivot(tNow := tr, tTotal := 1.0, pivot => pvt);		
		FOR i:=0 TO 1 DO
			FOR j:=0 TO 2 DO
				FlegRotA_FJntRef[i].data[j]:=(1-pvt)*FlegRotA_FJntState2[i,j]+pvt*(FlegRotA_FJntState3[i,j]);
			END_FOR
			gvl.legCtrl[Mapping23[i]].ForwardKinetics(motorAngles:=FlegRotA_FJntRef[i].data , legIndex:=Mapping23[i] , tipPosition=>FlegRotA_FPosWrtHip[i].data );
			fbRotMat(yaw := body_ref_ang_enter.data[2], pitch := body_ref_ang_enter.data[1],roll := body_ref_ang_enter.data[0], rm =>  Rb_target1 );
			temp.data[0]:=hip_pos[Mapping23[i],0];temp.data[1]:=hip_pos[Mapping23[i],1];temp.data[2]:=hip_pos[Mapping23[i],2];
			leg_ref_pos[Mapping23[i]]:= VecAdd( MatMulVec(Rb_target1, VecAdd(temp,MatMulVec(Rleg[Mapping23[i]],FlegRotA_FPosWrtHip[i]))),body_ref_pos);	
		END_FOR		
	ELSE		
		FlegRotAFinished:=TRUE;
		RequireReduceHeight:=TRUE;//***********************************************************************************************
	END_IF
END_IF
END_METHOD

METHOD PUBLIC TrjPlanning_FlegRotB : BOOL
VAR_INPUT
END_VAR
VAR
	FlegRotB_FJntState1:ARRAY[0..1,0..2] OF LREAL:=[0*pi/180,(162+1)*pi/180,172*pi/180,
                                                    0*pi/180,(162+1)*pi/180,172*pi/180];	//side rotates to horizon	
	FlegRotB_FJntState2:ARRAY[0..1,0..2] OF LREAL:=[0*pi/180,(162+1)*pi/180,81.588*pi/180,
                                                    0*pi/180,(162+1)*pi/180,81.588*pi/180];	;	//shank rotates to rc position
	(*FlegRotB_FJntState3:ARRAY[0..1,0..2] OF LREAL:=[0*pi/180,187.8384*pi/180,81.588*pi/180,
                                                    0*pi/180,187.8384*pi/180,81.588*pi/180];	//thigh rotates to RC position	[-0.3,-0.3209,-0.1246]*)
	FlegRotB_FJntState3Ref:ARRAY[0..1,0..2] OF LREAL:=[0*pi/180,222.0252*pi/180,(254.0072-222.0252)*pi/180,
                                                    0*pi/180,222.0252*pi/180,(254.0072-222.0252)*pi/180];	//thigh rotates to RC position	
	FlegRotB_FPosState3:ARRAY[0..1,0..2] OF LREAL:=[-0.15,-0.4-0.07,-0.1246,
													-0.15,-0.4-0.07,0.1246];	//thigh rotates to RC position													

																								 									 
	State1Time:LREAL:=1;
	State2Time:LREAL:=1;
	State3Time:LREAL:=1;
	State4Time:LREAL:=1;													 
													 
	tr: lreal;
	i: INT;
	j: INT;
	Rb_target1: Mat3;
	temp: vec3;
	tempLeg:ARRAY [0..2] OF LREAL;
	tempJnt:ARRAY [0..2] OF LREAL;
	tempRef:ARRAY [0..2] OF LREAL;
END_VAR
IF(gait_cycle-EnterFlegRotBCount)=1 THEN
	FOR i:=0 TO 1 DO
		tempLeg[0]:=FlegRotB_FPosState3[i,0];tempLeg[1]:=FlegRotB_FPosState3[i,1];tempLeg[2]:=FlegRotB_FPosState3[i,2];
		tempRef[0]:=FlegRotB_FJntState3Ref[i,0];tempRef[1]:=FlegRotB_FJntState3Ref[i,1];tempRef[2]:=FlegRotB_FJntState3Ref[i,2];
		GVL.legCtrl[Mapping23[i]].InverseKinetics(tipPosition:=tempLeg , refPosLast:=tempRef , legIndex:=Mapping23[i] , motorAngles=>tempJnt , isSingular=> );
		FlegRotB_FJntState3[i,0]:=tempJnt[0];FlegRotB_FJntState3[i,1]:=tempJnt[1];FlegRotB_FJntState3[i,2]:=tempJnt[2];
	END_FOR
END_IF

IF FlegRotBFinished=FALSE THEN
	IF(gait_cycle-EnterFlegRotBCount)<=State1Time*gvl.sampleRate THEN
		body_ref_pos:=body_ref_pos_enter;
		body_ref_ang:=body_ref_ang_enter;
		leg_ref_pos:=leg_ref_pos_enter;	
		
		tr  := UDINT_TO_LREAL(gait_cycle - EnterFlegRotBCount) / gvl.sampleRate / State1Time;
		fbGetPivot(tNow := tr, tTotal := 1.0, pivot => pvt);	
		FOR i:=0 TO 1 DO
			FOR j:=0 TO 2 DO
				FlegRotB_FJntRef[i].data[j]:=(1-pvt)*FlegRotB_FJntStart[i].data[j]+pvt*(FlegRotB_FJntState1[i,j]);
			END_FOR
			gvl.legCtrl[Mapping23[i]].ForwardKinetics(motorAngles:=FlegRotB_FJntRef[i].data , legIndex:=Mapping23[i] , tipPosition=>FlegRotB_FPosWrtHip[i].data );
			fbRotMat(yaw := body_ref_ang_enter.data[2], pitch := body_ref_ang_enter.data[1],roll := body_ref_ang_enter.data[0], rm =>  Rb_target1 );
			temp.data[0]:=hip_pos[Mapping23[i],0];temp.data[1]:=hip_pos[Mapping23[i],1];temp.data[2]:=hip_pos[Mapping23[i],2];
			leg_ref_pos[Mapping23[i]]:= VecAdd( MatMulVec(Rb_target1, VecAdd(temp,MatMulVec(Rleg[Mapping23[i]],FlegRotB_FPosWrtHip[i]))),body_ref_pos);	
		END_FOR
		
	ELSIF (gait_cycle-EnterFlegRotBCount)<=(State1Time+State2Time)*gvl.sampleRate THEN
		body_ref_pos:=body_ref_pos_enter;
		body_ref_ang:=body_ref_ang_enter;
		leg_ref_pos:=leg_ref_pos_enter;	
		
		tr  := (UDINT_TO_LREAL(gait_cycle - EnterFlegRotBCount) / gvl.sampleRate-State1Time) / State2Time;
		fbGetPivot(tNow := tr, tTotal := 1.0, pivot => pvt);	
		FOR i:=0 TO 1 DO
			FOR j:=0 TO 2 DO
				FlegRotB_FJntRef[i].data[j]:=(1-pvt)*FlegRotB_FJntState1[i,j]+pvt*(FlegRotB_FJntState2[i,j]);
			END_FOR
			gvl.legCtrl[Mapping23[i]].ForwardKinetics(motorAngles:=FlegRotB_FJntRef[i].data , legIndex:=Mapping23[i] , tipPosition=>FlegRotB_FPosWrtHip[i].data );
			fbRotMat(yaw := body_ref_ang_enter.data[2], pitch := body_ref_ang_enter.data[1],roll := body_ref_ang_enter.data[0], rm =>  Rb_target1 );
			temp.data[0]:=hip_pos[Mapping23[i],0];temp.data[1]:=hip_pos[Mapping23[i],1];temp.data[2]:=hip_pos[Mapping23[i],2];
			leg_ref_pos[Mapping23[i]]:= VecAdd( MatMulVec(Rb_target1, VecAdd(temp,MatMulVec(Rleg[Mapping23[i]],FlegRotB_FPosWrtHip[i]))),body_ref_pos);	
		END_FOR	
	ELSIF	(gait_cycle-EnterFlegRotBCount)<=(State1Time+State2Time+State3Time)*gvl.sampleRate THEN
		body_ref_pos:=body_ref_pos_enter;
		body_ref_ang:=body_ref_ang_enter;
		leg_ref_pos:=leg_ref_pos_enter;	
		tr  := (UDINT_TO_LREAL(gait_cycle - EnterFlegRotBCount) / gvl.sampleRate-State1Time-State2Time) / State3Time;
		fbGetPivot(tNow := tr, tTotal := 1.0, pivot => pvt);		
		FOR i:=0 TO 1 DO
			FOR j:=0 TO 2 DO
				FlegRotB_FJntRef[i].data[j]:=(1-pvt)*FlegRotB_FJntState2[i,j]+pvt*(FlegRotB_FJntState3[i,j]);
			END_FOR
			gvl.legCtrl[Mapping23[i]].ForwardKinetics(motorAngles:=FlegRotB_FJntRef[i].data , legIndex:=Mapping23[i] , tipPosition=>FlegRotB_FPosWrtHip[i].data );
			fbRotMat(yaw := body_ref_ang_enter.data[2], pitch := body_ref_ang_enter.data[1],roll := body_ref_ang_enter.data[0], rm =>  Rb_target1 );
			temp.data[0]:=hip_pos[Mapping23[i],0];temp.data[1]:=hip_pos[Mapping23[i],1];temp.data[2]:=hip_pos[Mapping23[i],2];
			leg_ref_pos[Mapping23[i]]:= VecAdd( MatMulVec(Rb_target1, VecAdd(temp,MatMulVec(Rleg[Mapping23[i]],FlegRotB_FPosWrtHip[i]))),body_ref_pos);	
		END_FOR			
	ELSE		
		FlegRotBFinished:=TRUE;
		RequireRecovery:=TRUE;//****************************************************************************************************
	END_IF
END_IF


(*IF FlegRotBFinished=FALSE AND (gait_cycle-EnterFlegRotBCount)<=FlegRotBTime*gvl.sampleRate THEN
	body_ref_pos:=body_ref_pos_enter;
	body_ref_ang:=body_ref_ang_enter;
	leg_ref_pos:=leg_ref_pos_enter;
	
	tr  := UDINT_TO_LREAL(gait_cycle - EnterFlegRotBCount) / gvl.sampleRate / FlegRotBTime;
	fbGetPivot(tNow := tr, tTotal := 1.0, pivot => pvt);
	FOR i:=0 TO 1 DO
		FOR j:=0 TO 2 DO
			FlegRotB_FJntRef[i].data[j]:=(1-pvt)*FlegRotB_FJntStart[i].data[j]+pvt*(FlegRotB_FJntTarget[i,j]);
		END_FOR
		gvl.legCtrl[Mapping23[i]].ForwardKinetics(motorAngles:=FlegRotB_FJntRef[i].data , legIndex:=Mapping23[i] , tipPosition=>FlegRotB_FPosWrtHip[i].data );
		fbRotMat(yaw := body_ref_ang_enter.data[2], pitch := body_ref_ang_enter.data[1],roll := body_ref_ang_enter.data[0], rm =>  Rb_target1 );
		temp.data[0]:=hip_pos[Mapping23[i],0];temp.data[1]:=hip_pos[Mapping23[i],1];temp.data[2]:=hip_pos[Mapping23[i],2];
		leg_ref_pos[Mapping23[i]]:= VecAdd( MatMulVec(Rb_target1, VecAdd(temp,MatMulVec(Rleg[Mapping23[i]],FlegRotB_FPosWrtHip[i]))),body_ref_pos);
	END_FOR
ELSE	
	FlegRotBFinished:=TRUE;
END_IF	*)
END_METHOD

METHOD PUBLIC TrjPlanning_LiftMleg : BOOL
VAR_INPUT
END_VAR

VAR
	tr: LREAL;
	i: INT;
	j: INT;
	Rb_target1: Mat3;
	temp: vec3;
END_VAR
IF LiftMlegFinished=FALSE AND (gait_cycle-EnterLiftMlegCount)<=LiftMlegTime*gvl.sampleRate THEN
	body_ref_pos:=body_ref_pos_enter;
	body_ref_ang:=body_ref_ang_enter;
	leg_ref_pos:=leg_ref_pos_enter;
	tr  := UDINT_TO_LREAL(gait_cycle - EnterLiftMlegCount) / gvl.sampleRate / LiftMlegTime;
	fbGetPivot(tNow := tr, tTotal := 1.0, pivot => pvt);
	FOR i:=0 TO 1 DO
		LiftMleg_MJntRef[i]:=LiftMleg_MJntStart[i];
		LiftMleg_MJntRef[i].data[2]:=(1-pvt)*LiftMleg_MJntStart[i].data[2]+pvt*(LiftMleg_MJntStart[i].data[2]-5*pi/180);
	
	gvl.legCtrl[Mapping14[i]].ForwardKinetics(motorAngles:=LiftMleg_MJntRef[i].data , legIndex:=Mapping14[i] , tipPosition=>LiftMleg_MPosWrtHip[i].data );
	fbRotMat(yaw := body_ref_ang_enter.data[2], pitch := body_ref_ang_enter.data[1],roll := body_ref_ang_enter.data[0], rm =>  Rb_target1 );
	temp.data[0]:=hip_pos[Mapping14[i],0];temp.data[1]:=hip_pos[Mapping14[i],1];temp.data[2]:=hip_pos[Mapping14[i],2];
	leg_ref_pos[Mapping14[i]]:= VecAdd( MatMulVec(Rb_target1, VecAdd(temp,MatMulVec(Rleg[Mapping14[i]],LiftMleg_MPosWrtHip[i]))),body_ref_pos);
	END_FOR
ELSE
	LiftMlegFinished:=TRUE;
END_IF
END_METHOD

METHOD PUBLIC TrjPlanning_MlegRollA : BOOL
VAR_INPUT
	
END_VAR

VAR
	MlegRollA_MPosTarget:ARRAY[0..1,0..2] OF LREAL:=[-0.2,-0.4-0.07,-0.1246,
                                                     -0.2,-0.4-0.07,0.1246];													 
	MlegRollA_MJntTargetRef:ARRAY[0..1,0..2] OF LREAL:=[0,579.7161*pi/180,-303.4078*pi/180,
                                                     0,579.7161*pi/180,-303.4078*pi/180];	//invert rotation for shank and thigh, [-0.2,-0.4-0.07,-0.1246]
										 
	tr: lreal;
	i: INT;
	j: INT;
	Rb_target1: Mat3;
	temp: vec3;
	tempLeg:ARRAY [0..2] OF LREAL;
	tempJnt:ARRAY [0..2] OF LREAL;
	tempRef:ARRAY [0..2] OF LREAL;
	
	tipForceDesireLegAF:	 ARRAY[0..5,0..2] OF LREAL:=[0,-100,0,
													 0,0,0,
													 0,0,0,
													 0,0,0,
													 0,0,0,
													 0,-120,0];
END_VAR
IF (gait_cycle-EnterMlegRollACount)=1 THEN
	FOR i:=0 TO 1 DO
		tempLeg[0]:=MlegRollA_MPosTarget[i,0];tempLeg[1]:=MlegRollA_MPosTarget[i,1];tempLeg[2]:=MlegRollA_MPosTarget[i,2];
		tempRef[0]:=MlegRollA_MJntTargetRef[i,0];tempRef[1]:=MlegRollA_MJntTargetRef[i,1];tempRef[2]:=MlegRollA_MJntTargetRef[i,2];
		GVL.legCtrl[Mapping14[i]].InverseKinetics(tipPosition:=tempLeg , refPosLast:=tempRef , legIndex:=Mapping14[i] , motorAngles=>tempJnt , isSingular=> );
		MlegRollA_MJntTarget[i,0]:=tempJnt[0];MlegRollA_MJntTarget[i,1]:=tempJnt[1];MlegRollA_MJntTarget[i,2]:=tempJnt[2];		
	END_FOR
END_IF

IF MlegRollAFinished=FALSE AND (gait_cycle-EnterMlegRollACount)<=MlegRollATime*gvl.sampleRate THEN
	body_ref_pos:=body_ref_pos_enter;
	body_ref_ang:=body_ref_ang_enter;
	leg_ref_pos:=leg_ref_pos_enter;
	
	tr  := UDINT_TO_LREAL(gait_cycle - EnterMlegRollACount) / gvl.sampleRate / MlegRollATime;
	fbGetPivot(tNow := tr, tTotal := 1.0, pivot => pvt);
	FOR i:=0 TO 1 DO
		FOR j:=0 TO 2 DO
			MlegRollA_MJntRef[i].data[j]:=(1-pvt)*MlegRollA_MJntStart[i].data[j]+pvt*(MlegRollA_MJntTarget[i,j]);
		END_FOR
		gvl.legCtrl[Mapping14[i]].ForwardKinetics(motorAngles:=MlegRollA_MJntRef[i].data , legIndex:=Mapping14[i] , tipPosition=>MlegRollA_MPosWrtHip[i].data );
		fbRotMat(yaw := body_ref_ang_enter.data[2], pitch := body_ref_ang_enter.data[1],roll := body_ref_ang_enter.data[0], rm =>  Rb_target1 );
		temp.data[0]:=hip_pos[Mapping14[i],0];temp.data[1]:=hip_pos[Mapping14[i],1];temp.data[2]:=hip_pos[Mapping14[i],2];
		leg_ref_pos[Mapping14[i]]:= VecAdd( MatMulVec(Rb_target1, VecAdd(temp,MatMulVec(Rleg[Mapping14[i]],MlegRollA_MPosWrtHip[i]))),body_ref_pos);
	END_FOR
	
	//force compensator
	tipForceTarget:=tipForceDesireLegAF;
	IF (gait_cycle-EnterMlegRollACount)<=fceLoadTime*gvl.sampleRate THEN
		tr  := UDINT_TO_LREAL(gait_cycle-EnterMlegRollACount) / gvl.sampleRate / fceLoadTime;
		fbGetPivot(tNow := tr, tTotal := 1.0, pivot => pvt);
		FOR i:=0 TO 5 DO
			FOR j:=0 TO 2 DO
				tipForceDesire[i,j]:=(1-pvt)*tipForceDesireZeros[i,j]+pvt*tipForceTarget[i,j];
			END_FOR
		END_FOR
	ELSIF (gait_cycle-EnterMlegRollACount)>(MlegRollATime-fceLoadTime)*gvl.sampleRate AND (gait_cycle-EnterMlegRollACount)<=MlegRollATime*gvl.sampleRate THEN
		tr  := (UDINT_TO_LREAL(gait_cycle-EnterMlegRollACount) / gvl.sampleRate -(MlegRollATime-fceLoadTime))/ fceLoadTime;
		fbGetPivot(tNow := tr, tTotal := 1.0, pivot => pvt);
		FOR i:=0 TO 5 DO
			FOR j:=0 TO 2 DO
				tipForceDesire[i,j]:=(1-pvt)*tipForceTarget[i,j]+pvt*tipForceDesireZeros[i,j];
			END_FOR
		END_FOR	
	END_IF
					
ELSE	
	MlegRollAFinished:=TRUE;
	tipForceDesire:=tipForceDesireZeros;
	RequireFlegRotA:=TRUE;//*******************************************************************************************************
END_IF
END_METHOD

METHOD PUBLIC TrjPlanning_MlegRollB : BOOL
VAR_INPUT
END_VAR
VAR
	MlegRollB_MPosTarget:ARRAY[0..1,0..2] OF LREAL:=[-0.0141,-0.1797,-0.1246,
                                                     -0.0141,-0.1797,0.1246];
	MlegRollB_MJntTargetRef:ARRAY[0..1,0..2] OF LREAL:=[0,331.45*pi/180,-144*pi/180,
                                                     0,331.45*pi/180,-144*pi/180];//invert rotation for shank and thigh, old version
												 							 
	tr: LREAL;
	i: INT;
	j: INT;
	Rb_target1: Mat3;
	temp: vec3;
	tempLeg:ARRAY [0..2] OF LREAL;
	tempJnt:ARRAY [0..2] OF LREAL;
	tempRef:ARRAY [0..2] OF LREAL;	
	
	tipForceDesireLegAF:	 ARRAY[0..5,0..2] OF LREAL:=[0,0,0,
													 0,0,0,
													 0,0,0,
													 0,0,0,
													 0,0,0,
													 0,0,0];//-100,-120
END_VAR
IF (gait_cycle-EnterMlegRollBCount)=1 THEN
	FOR i:=0 TO 1 DO
		tempLeg[0]:=MlegRollB_MPosTarget[i,0];tempLeg[1]:=MlegRollB_MPosTarget[i,1];tempLeg[2]:=MlegRollB_MPosTarget[i,2];
		tempRef[0]:=MlegRollB_MJntTargetRef[i,0];tempRef[1]:=MlegRollB_MJntTargetRef[i,1];tempRef[2]:=MlegRollB_MJntTargetRef[i,2];
		GVL.legCtrl[Mapping14[i]].InverseKinetics(tipPosition:=tempLeg , refPosLast:=tempRef , legIndex:=Mapping14[i] , motorAngles=>tempJnt , isSingular=> );
		MlegRollB_MJntTarget[i,0]:=tempJnt[0];MlegRollB_MJntTarget[i,1]:=tempJnt[1];MlegRollB_MJntTarget[i,2]:=tempJnt[2];		
	END_FOR
END_IF

IF MlegRollBFinished=FALSE AND (gait_cycle-EnterMlegRollBCount)<=MlegRollBTime*gvl.sampleRate THEN
	body_ref_pos:=body_ref_pos_enter;
	body_ref_ang:=body_ref_ang_enter;
	leg_ref_pos:=leg_ref_pos_enter;
	tr  := UDINT_TO_LREAL(gait_cycle - EnterMlegRollBCount) / gvl.sampleRate / MlegRollBTime;
	fbGetPivot(tNow := tr, tTotal := 1.0, pivot => pvt);
	FOR i:=0 TO 1 DO
		FOR j:=0 TO 2 DO
			MlegRollB_MJntRef[i].data[j]:=(1-pvt)*MlegRollB_MJntStart[i].data[j]+pvt*(MlegRollB_MJntTarget[i,j]);
		END_FOR
		gvl.legCtrl[Mapping14[i]].ForwardKinetics(motorAngles:=MlegRollB_MJntRef[i].data , legIndex:=Mapping14[i] , tipPosition=>MlegRollB_MPosWrtHip[i].data );
		fbRotMat(yaw := body_ref_ang_enter.data[2], pitch := body_ref_ang_enter.data[1],roll := body_ref_ang_enter.data[0], rm =>  Rb_target1 );
		temp.data[0]:=hip_pos[Mapping14[i],0];temp.data[1]:=hip_pos[Mapping14[i],1];temp.data[2]:=hip_pos[Mapping14[i],2];
		leg_ref_pos[Mapping14[i]]:= VecAdd( MatMulVec(Rb_target1, VecAdd(temp,MatMulVec(Rleg[Mapping14[i]],MlegRollB_MPosWrtHip[i]))),body_ref_pos);
	END_FOR
	
	//force compensator
	tipForceTarget:=tipForceDesireLegAF;
	IF (gait_cycle-EnterMlegRollBCount)<=fceLoadTime*gvl.sampleRate THEN
		tr  := UDINT_TO_LREAL(gait_cycle-EnterMlegRollBCount) / gvl.sampleRate / fceLoadTime;
		fbGetPivot(tNow := tr, tTotal := 1.0, pivot => pvt);
		FOR i:=0 TO 5 DO
			FOR j:=0 TO 2 DO
				tipForceDesire[i,j]:=(1-pvt)*tipForceDesireZeros[i,j]+pvt*tipForceTarget[i,j];
			END_FOR
		END_FOR
	ELSIF (gait_cycle-EnterMlegRollBCount)>(MlegRollBTime-fceLoadTime)*gvl.sampleRate AND (gait_cycle-EnterMlegRollBCount)<=MlegRollBTime*gvl.sampleRate THEN
		tr  := (UDINT_TO_LREAL(gait_cycle-EnterMlegRollBCount) / gvl.sampleRate -(MlegRollBTime-fceLoadTime))/ fceLoadTime;
		fbGetPivot(tNow := tr, tTotal := 1.0, pivot => pvt);
		FOR i:=0 TO 5 DO
			FOR j:=0 TO 2 DO
				tipForceDesire[i,j]:=(1-pvt)*tipForceTarget[i,j]+pvt*tipForceDesireZeros[i,j];
			END_FOR
		END_FOR	
	END_IF	
	
ELSE	
	MlegRollBFinished:=TRUE;
	tipForceDesire:=tipForceDesireZeros;
END_IF
END_METHOD

METHOD PUBLIC TrjPlanning_MlegRollC : BOOL
VAR_INPUT
END_VAR
VAR
	MlegRollC_MPosTarget:ARRAY[0..1,0..2] OF LREAL:=[-0.2,-0.1797,-0.1246,
                                                     -0.2,-0.1797,0.1246];
	MlegRollC_MJntTargetRef:ARRAY[0..1,0..2] OF LREAL:=[0,523.2736*pi/180,-235.1052*pi/180,
                                                     0,523.2736*pi/180,-235.1052*pi/180];//invert rotation for shank and thigh, a more rotation for shank, old version										 
													 
	tr: lreal;
	i: INT;
	j: INT;
	Rb_target1: Mat3;
	temp: vec3;
	tempLeg:ARRAY [0..2] OF LREAL;
	tempJnt:ARRAY [0..2] OF LREAL;
	tempRef:ARRAY [0..2] OF LREAL;	
	
	tipForceDesireLegAF:	 ARRAY[0..5,0..2] OF LREAL:=[0,-100,0,
													 0,0,0,
													 0,0,0,
													 0,0,0,
													 0,0,0,
													 0,-120,0];
END_VAR
IF (gait_cycle-EnterMlegRollCCount)=1 THEN
	FOR i:=0 TO 1 DO
		tempLeg[0]:=MlegRollC_MPosTarget[i,0];tempLeg[1]:=MlegRollC_MPosTarget[i,1];tempLeg[2]:=MlegRollC_MPosTarget[i,2];
		tempRef[0]:=MlegRollC_MJntTargetRef[i,0];tempRef[1]:=MlegRollC_MJntTargetRef[i,1];tempRef[2]:=MlegRollC_MJntTargetRef[i,2];
		GVL.legCtrl[Mapping14[i]].InverseKinetics(tipPosition:=tempLeg , refPosLast:=tempRef , legIndex:=Mapping14[i] , motorAngles=>tempJnt , isSingular=> );
		MlegRollC_MJntTarget[i,0]:=tempJnt[0];MlegRollC_MJntTarget[i,1]:=tempJnt[1];MlegRollC_MJntTarget[i,2]:=tempJnt[2];		
	END_FOR
END_IF

IF MlegRollCFinished=FALSE AND (gait_cycle-EnterMlegRollCCount)<=MlegRollCTime*gvl.sampleRate THEN
	body_ref_pos:=body_ref_pos_enter;
	body_ref_ang:=body_ref_ang_enter;
	leg_ref_pos:=leg_ref_pos_enter;
	
	tr  := UDINT_TO_LREAL(gait_cycle - EnterMlegRollCCount) / gvl.sampleRate / MlegRollCTime;
	fbGetPivot(tNow := tr, tTotal := 1.0, pivot => pvt);
	FOR i:=0 TO 1 DO
		FOR j:=0 TO 2 DO
			MlegRollC_MJntRef[i].data[j]:=(1-pvt)*MlegRollC_MJntStart[i].data[j]+pvt*(MlegRollC_MJntTarget[i,j]);
		END_FOR
		gvl.legCtrl[Mapping14[i]].ForwardKinetics(motorAngles:=MlegRollC_MJntRef[i].data , legIndex:=Mapping14[i] , tipPosition=>MlegRollC_MPosWrtHip[i].data );
		fbRotMat(yaw := body_ref_ang_enter.data[2], pitch := body_ref_ang_enter.data[1],roll := body_ref_ang_enter.data[0], rm =>  Rb_target1 );
		temp.data[0]:=hip_pos[Mapping14[i],0];temp.data[1]:=hip_pos[Mapping14[i],1];temp.data[2]:=hip_pos[Mapping14[i],2];
		leg_ref_pos[Mapping14[i]]:= VecAdd( MatMulVec(Rb_target1, VecAdd(temp,MatMulVec(Rleg[Mapping14[i]],MlegRollC_MPosWrtHip[i]))),body_ref_pos);
	END_FOR	
	
	//force compensator
	tipForceTarget:=tipForceDesireLegAF;
	IF (gait_cycle-EnterMlegRollCCount)<=fceLoadTime*gvl.sampleRate THEN
		tr  := UDINT_TO_LREAL(gait_cycle-EnterMlegRollCCount) / gvl.sampleRate / fceLoadTime;
		fbGetPivot(tNow := tr, tTotal := 1.0, pivot => pvt);
		FOR i:=0 TO 5 DO
			FOR j:=0 TO 2 DO
				tipForceDesire[i,j]:=(1-pvt)*tipForceDesireZeros[i,j]+pvt*tipForceTarget[i,j];
			END_FOR
		END_FOR
	ELSIF (gait_cycle-EnterMlegRollCCount)>(MlegRollCTime-fceLoadTime)*gvl.sampleRate AND (gait_cycle-EnterMlegRollCCount)<=MlegRollCTime*gvl.sampleRate THEN
		tr  := (UDINT_TO_LREAL(gait_cycle-EnterMlegRollCCount) / gvl.sampleRate -(MlegRollCTime-fceLoadTime))/ fceLoadTime;
		fbGetPivot(tNow := tr, tTotal := 1.0, pivot => pvt);
		FOR i:=0 TO 5 DO
			FOR j:=0 TO 2 DO
				tipForceDesire[i,j]:=(1-pvt)*tipForceTarget[i,j]+pvt*tipForceDesireZeros[i,j];
			END_FOR
		END_FOR	
	END_IF
	
ELSE	
	MlegRollCFinished:=TRUE;
	tipForceDesire:=tipForceDesireZeros;
	RequireAddHeight:=TRUE;//*******************************************************************************************************
END_IF
END_METHOD

METHOD PUBLIC TrjPlanning_OrientAdjust : BOOL
VAR_INPUT
END_VAR

VAR
	tr: LREAL;
	i: INT;
	Rb_target1: Mat3;
	temp: VEC3;
	j: INT;
	(*OA_MJntExtend:ARRAY[0..1,0..2] OF LREAL:=[0,331.45*pi/180,-144*pi/180,
                                                     0,331.45*pi/180,-144*pi/180];
	OA_MJntExtract:ARRAY[0..1,0..2] OF LREAL:=[0,340*pi/180,-155*pi/180,
                                                     0,340*pi/180,-155*pi/180];*)
END_VAR
IF OrientAdjustFinished=FALSE AND (gait_cycle-EnterOrientAdjustCount)<=LREAL_TO_UDINT((2*OA_LiftGroundTime+OA_AdjustTime+OA_AdjustExtractTime+OA_AdjustExtendTime)*gvl.sampleRate) THEN
	IF (gait_cycle-EnterOrientAdjustCount)<=LREAL_TO_UDINT((OA_LiftGroundTime)*gvl.sampleRate) THEN
		leg_ref_pos:=leg_ref_pos_enter;
		body_ref_ang:=OA_BodyAngStart;
		body_ref_pos:=OA_BodyPosStart;
		tr  := UDINT_TO_LREAL(gait_cycle - EnterOrientAdjustCount) / gvl.sampleRate /OA_LiftGroundTime;
		fbGetPivot(tNow := tr, tTotal := 1.0, pivot => pvt);	
		body_ref_pos.data[2]:=(1-pvt)*OA_BodyPosStart.data[2]+pvt*(OA_BodyPosStart.data[2]+OA_HeighAdd);
		FOR i:=0 TO 1 DO
			gvl.legCtrl[Mapping23[i]].ForwardKinetics(motorAngles:=OA_FJntRef[i].data , legIndex:=Mapping23[i] , tipPosition=>OA_FPosWrtHip[i].data );
			fbRotMat(yaw := body_ref_ang.data[2], pitch := body_ref_ang.data[1],roll := body_ref_ang.data[0], rm =>  Rb_target1 );
			temp.data[0]:=hip_pos[Mapping23[i],0];temp.data[1]:=hip_pos[Mapping23[i],1];temp.data[2]:=hip_pos[Mapping23[i],2];
			leg_ref_pos[Mapping23[i]]:= VecAdd( MatMulVec(Rb_target1, VecAdd(temp,MatMulVec(Rleg[Mapping23[i]],OA_FPosWrtHip[i]))),body_ref_pos);			
		END_FOR
	ELSIF (gait_cycle-EnterOrientAdjustCount)<=LREAL_TO_UDINT((OA_LiftGroundTime+OA_AdjustTime)*gvl.sampleRate) THEN
		leg_ref_pos:=leg_ref_pos_enter;
		tr  := (UDINT_TO_LREAL(gait_cycle - EnterOrientAdjustCount) / gvl.sampleRate -OA_LiftGroundTime)/OA_AdjustTime;
		fbGetPivot(tNow := tr, tTotal := 1.0, pivot => pvt);
		FOR i:=0 TO 2 DO
			body_ref_pos.data[i]:=(1-pvt)*OA_BodyPosStart.data[i]+pvt*OA_BodyPoseEnd.data[i];
			body_ref_ang.data[i]:=(1-pvt)*OA_BodyAngStart.data[i]+pvt*OA_BodyAngEnd.data[i];
		END_FOR		
		body_ref_pos.data[2]:=body_ref_pos.data[2]+OA_HeighAdd;
		FOR i:=0 TO 1 DO
			gvl.legCtrl[Mapping23[i]].ForwardKinetics(motorAngles:=OA_FJntRef[i].data , legIndex:=Mapping23[i] , tipPosition=>OA_FPosWrtHip[i].data );
			fbRotMat(yaw := body_ref_ang.data[2], pitch := body_ref_ang.data[1],roll := body_ref_ang.data[0], rm =>  Rb_target1 );
			temp.data[0]:=hip_pos[Mapping23[i],0];temp.data[1]:=hip_pos[Mapping23[i],1];temp.data[2]:=hip_pos[Mapping23[i],2];
			leg_ref_pos[Mapping23[i]]:= VecAdd( MatMulVec(Rb_target1, VecAdd(temp,MatMulVec(Rleg[Mapping23[i]],OA_FPosWrtHip[i]))),body_ref_pos);			
		END_FOR
	ELSIF (gait_cycle-EnterOrientAdjustCount)<=LREAL_TO_UDINT((2*OA_LiftGroundTime+OA_AdjustTime)*gvl.sampleRate) THEN	
		leg_ref_pos:=leg_ref_pos_enter;
		body_ref_ang:=OA_BodyAngEnd;
		body_ref_pos:=OA_BodyPoseEnd;
		tr  := (UDINT_TO_LREAL(gait_cycle - EnterOrientAdjustCount) / gvl.sampleRate-OA_LiftGroundTime-OA_AdjustTime )/OA_LiftGroundTime;
		fbGetPivot(tNow := tr, tTotal := 1.0, pivot => pvt);	
		body_ref_pos.data[2]:=(1-pvt)*(OA_BodyPosStart.data[2]+OA_HeighAdd)+pvt*OA_BodyPosStart.data[2];
		FOR i:=0 TO 1 DO
			gvl.legCtrl[Mapping23[i]].ForwardKinetics(motorAngles:=OA_FJntRef[i].data , legIndex:=Mapping23[i] , tipPosition=>OA_FPosWrtHip[i].data );
			fbRotMat(yaw := body_ref_ang.data[2], pitch := body_ref_ang.data[1],roll := body_ref_ang.data[0], rm =>  Rb_target1 );
			temp.data[0]:=hip_pos[Mapping23[i],0];temp.data[1]:=hip_pos[Mapping23[i],1];temp.data[2]:=hip_pos[Mapping23[i],2];
			leg_ref_pos[Mapping23[i]]:= VecAdd( MatMulVec(Rb_target1, VecAdd(temp,MatMulVec(Rleg[Mapping23[i]],OA_FPosWrtHip[i]))),body_ref_pos);			
		END_FOR		
		IF (gait_cycle-EnterOrientAdjustCount)=LREAL_TO_UDINT((2*OA_LiftGroundTime+OA_AdjustTime)*gvl.sampleRate) THEN
			OA_legPosEnterExtract:=leg_ref_pos;
			FOR i:=0 TO 1 DO
				FOR j:=0 TO 2 DO
					OA_MJntStart[i].data[j]:=jointPosLast[Mapping14[i],j];
				END_FOR
			END_FOR			
		END_IF
	ELSIF (gait_cycle-EnterOrientAdjustCount)<=LREAL_TO_UDINT((2*OA_LiftGroundTime+OA_AdjustTime+OA_AdjustExtractTime)*gvl.sampleRate) THEN	
		body_ref_pos:=OA_BodyPoseEnd;
		body_ref_ang:=OA_BodyAngEnd;
		leg_ref_pos:=OA_legPosEnterExtract;
		tr  := (UDINT_TO_LREAL(gait_cycle - EnterOrientAdjustCount) / gvl.sampleRate-2*OA_LiftGroundTime-OA_AdjustTime )/OA_AdjustExtractTime;
		fbGetPivot(tNow := tr, tTotal := 1.0, pivot => pvt);	
		FOR i:=0 TO 1 DO
			FOR j:=0 TO 2 DO
				OA_MJntRef[i].data[j]:=(1-pvt)*OA_MJntStart[i].data[j]+pvt*OA_MJntExtract[i,j];
			END_FOR
			gvl.legCtrl[Mapping14[i]].ForwardKinetics(motorAngles:=OA_MJntRef[i].data , legIndex:=Mapping14[i] , tipPosition=>OA_MPosWrtHip[i].data );
			fbRotMat(yaw := body_ref_ang.data[2], pitch := body_ref_ang.data[1],roll := body_ref_ang.data[0], rm =>  Rb_target1 );
			temp.data[0]:=hip_pos[Mapping14[i],0];temp.data[1]:=hip_pos[Mapping14[i],1];temp.data[2]:=hip_pos[Mapping14[i],2];
			leg_ref_pos[Mapping14[i]]:= VecAdd( MatMulVec(Rb_target1, VecAdd(temp,MatMulVec(Rleg[Mapping14[i]],OA_MPosWrtHip[i]))),body_ref_pos);
			
